Fanuc TP program (LS listing): MAKROSTP.LS

/PROG  MAKROSTP
/ATTR
OWNER		= MNEDITOR;
COMMENT		= "MAKRO_SCHRITT";
PROG_SIZE	= 100704;
CREATE		= DATE 11-01-11  TIME 07:00:00;
MODIFIED	= DATE 20-09-12  TIME 10:46:22;
FILE_NAME	= ;
VERSION		= 0;
LINE_COUNT	= 4405;
MEMORY_SIZE	= 103104;
PROTECT		= READ_WRITE;
TCD:  STACK_SIZE	= 0,
      TASK_PRIORITY	= 100,
      TIME_SLICE	= 0,
      BUSY_LAMP_OFF	= 1,
      ABORT_REQUEST	= 7,
      PAUSE_REQUEST	= 3;
DEFAULT_GROUP	= *,*,*,*,*;
CONTROL_CODE	= 00000000 00000010;
/MN
   1:  !Schrittkette Konzernstandard ;
   2:  !KS24 ;
   3:  !Version: 02 ;
   4:  !Stand: 003 MOD KN ;
   5:  !letzte Aenderung 30.07.2015 DB ;
   6:  !Mod von KN --> S2 mit Wartezeit ;
   7:   ;
   8:  !Zaehler [41] = aktueller Schritt ;
   9:  !Zaehler [42] = letzter Schritt ;
  10:  R[41]=0    ;
  11:  R[42]=0    ;
  12:   ;
  13:   ;
  14:  !*********************** ;
  15:  !*********************** ;
  16:  !* Start Makro_Schritt * ;
  17:  !*********************** ;
  18:  !*********************** ;
  19:   ;
  20:   ;
  21:  !***************************** ;
  22:  !*         Schritt 1         * ;
  23:  !* E/A's / Flags Ruecksetzen * ;
  24:  !***************************** ;
  25:   ;
  26:  !Loop fuer Schrittkette LBL[1] ;
  27:  LBL[1] ;
  28:  R[41]=1    ;
  29:  !Statusbildschirm einblenden ;
  30:  DO[18181]=(OFF) ;
  31:  !SK1 KF1 KS1 ;
  32:  DO[786]=(OFF) ;
  33:  DO[834]=(OFF) ;
  34:  DO[842]=(OFF) ;
  35:  DO[847]=(OFF) ;
  36:  !SK2 KF2 KS2 ;
  37:  DO[946]=(OFF) ;
  38:  DO[994]=(OFF) ;
  39:  DO[995]=(OFF) ;
  40:  DO[1002]=(OFF) ;
  41:  !SK3 KF3 KS3 ;
  42:  DO[1106]=(OFF) ;
  43:  DO[1154]=(OFF) ;
  44:  DO[1155]=(OFF) ;
  45:  DO[1162]=(OFF) ;
  46:  !KS1 KS2 KS3 ;
  47:  DO[3969]=(OFF) ;
  48:  DO[3970]=(OFF) ;
  49:  DO[3971]=(OFF) ;
  50:  !Auswahl EZ1/SP1 an KF2 ;
  51:  F[72]=(OFF) ;
  52:  !Auswahl EZ1/SP1 an KF3 ;
  53:  F[73]=(OFF) ;
  54:  !Auswert. KF Umdrehungen EZ1/SP1 ;
  55:  F[94]=(OFF) ;
  56:  F[95]=(OFF) ;
  57:  F[96]=(OFF) ;
  58:  F[97]=(OFF) ;
  59:  F[98]=(OFF) ;
  60:  F[99]=(OFF) ;
  61:  F[100]=(OFF) ;
  62:  F[101]=(OFF) ;
  63:  F[102]=(OFF) ;
  64:  F[103]=(OFF) ;
  65:  F[104]=(OFF) ;
  66:  F[105]=(OFF) ;
  67:  F[106]=(OFF) ;
  68:  F[107]=(OFF) ;
  69:  F[108]=(OFF) ;
  70:  F[109]=(OFF) ;
  71:  F[110]=(OFF) ;
  72:  F[111]=(OFF) ;
  73:  F[112]=(OFF) ;
  74:  F[113]=(OFF) ;
  75:  F[114]=(OFF) ;
  76:  F[115]=(OFF) ;
  77:  F[116]=(OFF) ;
  78:  F[117]=(OFF) ;
  79:  !Auswert. KF Umdrehungen EZ2/SP2 ;
  80:  F[150]=(OFF) ;
  81:  F[151]=(OFF) ;
  82:  F[152]=(OFF) ;
  83:  F[153]=(OFF) ;
  84:  F[154]=(OFF) ;
  85:  F[155]=(OFF) ;
  86:  !Auswert. KF Umdrehungen EZ3/SP3 ;
  87:  F[186]=(OFF) ;
  88:  F[187]=(OFF) ;
  89:  F[188]=(OFF) ;
  90:  F[189]=(OFF) ;
  91:  F[190]=(OFF) ;
  92:  F[191]=(OFF) ;
  93:  !Hilfsflags beim Fraesen ;
  94:  F[287]=(OFF) ;
  95:  F[290]=(OFF) ;
  96:  F[291]=(OFF) ;
  97:  F[301]=(OFF) ;
  98:  !Hilfsflags SZ2 an SK1 ;
  99:  F[307]=(OFF) ;
 100:  F[308]=(OFF) ;
 101:  !Hilfsflags KF Initiator ;
 102:  F[312]=(OFF) ;
 103:  F[313]=(OFF) ;
 104:  !RSK Fehlerausgaben ;
 105:  F[322]=(OFF) ;
 106:  F[323]=(OFF) ;
 107:  F[324]=(OFF) ;
 108:  F[325]=(OFF) ;
 109:  F[326]=(OFF) ;
 110:  F[327]=(OFF) ;
 111:  F[328]=(OFF) ;
 112:  F[329]=(OFF) ;
 113:  !Flag KL1 Spueleimer ;
 114:  F[352]=(OFF) ;
 115:  F[353]=(OFF) ;
 116:  !Flag KL2 Spueleimer ;
 117:  F[373]=(OFF) ;
 118:  F[374]=(OFF) ;
 119:  !Flag KL3 Spueleimer ;
 120:  F[394]=(OFF) ;
 121:  F[395]=(OFF) ;
 122:  !Flag MS Reinigung gestartet ;
 123:  F[604]=(OFF) ;
 124:  F[605]=(OFF) ;
 125:  F[608]=(OFF) ;
 126:  !Flag für Grundstellung RSK ;
 127:  F[321]=(OFF) ;
 128:  !Ruecksetzen Fraeszaehler ;
 129:  R[1]=0    ;
 130:  R[42]=1    ;
 131:  JMP LBL[2] ;
 132:   ;
 133:   ;
 134:  !************************ ;
 135:  !************************ ;
 136:  !* RSK in Grundstellung * ;
 137:  !************************ ;
 138:  !************************ ;
 139:   ;
 140:   ;
 141:  !*********************** ;
 142:  !*      Schritt 2      * ;
 143:  !* Funktionsauswertung * ;
 144:  !*********************** ;
 145:   ;
 146:  LBL[2] ;
 147:  R[41]=2    ;
 148:  F[321]=(ON) ;
 149:   ;
 150:  !Fraesen ROB EZ1/SP1 SZ1-SZ4 ;
 151:  !an KF1 ;
 152:  IF ((F[90] AND !F[91]) AND !F[72] AND !F[73] AND (F[64] OR F[65] OR F[66] OR F[67])),R[41]=3 ;
 153:   ;
 154:  !Fraesen ROB EZ1/SP1 SZ1-SZ4 ;
 155:  !an KF2 ;
 156:  IF ((F[90] AND !F[91]) AND F[72] AND !F[73] AND (F[64] OR F[65] OR F[66] OR F[67])),R[41]=58 ;
 157:   ;
 158:  !Fraesen ROB EZ1/SP1 SZ1-SZ4 ;
 159:  !an KF3 ;
 160:  IF ((F[90] AND !F[91]) AND !F[72] AND F[73] AND (F[64] OR F[65] OR F[66] OR F[67])),R[41]=64 ;
 161:   ;
 162:  !Fraesen STAT EZ1/SP1 ;
 163:  IF (F[92] AND !F[93]),R[41]=9 ;
 164:   ;
 165:  !Fraesen STAT EZ2/SP2 ;
 166:  IF (F[148] AND !F[149]),R[41]=18 ;
 167:   ;
 168:  !Fraesen STAT EZ3/SP3 ;
 169:  IF (F[184] AND !F[185]),R[41]=27 ;
 170:   ;
 171:  !MS1 Reinigung an KS3 ;
 172:  IF (F[603] AND !F[605] AND F[528] AND !F[529]),R[41]=36 ;
 173:   ;
 174:  !MS2 Reinigung an KS2 ;
 175:  IF (F[607] AND !F[609] AND F[528] AND !F[529]),R[41]=40 ;
 176:   ;
 177:  !KL1 Spueleimer (an Pneum. Schwen ;
 178:  !in Arbeitsstellung schwenken ;
 179:  IF (!F[352] AND F[353] AND !F[355] AND ((F[523] AND !F[524]) OR (!F[523] AND F[524]))),R[41]=44 ;
 180:   ;
 181:  !KL1 Spueleimer (an Pneum. Schwen ;
 182:  !in Ruhestellung schwenken ;
 183:  IF (F[352] AND !F[353] AND !F[355] AND ((F[523] AND !F[524]) OR (!F[523] AND F[524]))),R[41]=45 ;
 184:   ;
 185:  !KL2 Spueleimer (an Pneum. Schwen ;
 186:  !in Arbeitsstellung schwenken ;
 187:  IF (!F[373] AND F[374] AND !F[376] AND ((F[523] AND !F[524]) OR (!F[523] AND F[524]))),R[41]=46 ;
 188:   ;
 189:  !KL2 Spueleimer (an Pneum. Schwen ;
 190:  !in Ruhestellung schwenken ;
 191:  IF (F[373] AND !F[374] AND !F[376] AND ((F[523] AND !F[524]) OR (!F[523] AND F[524]))),R[41]=47 ;
 192:   ;
 193:  !KL3 Spueleimer (an Pneum. Schwen ;
 194:  !in Arbeitsstellung schwenken ;
 195:  IF (!F[394] AND F[395] AND !F[397] AND ((F[523] AND !F[524]) OR (!F[523] AND F[524]))),R[41]=48 ;
 196:   ;
 197:  !KL3 Spueleimer (an Pneum. Schwen ;
 198:  !in Ruhestellung schwenken ;
 199:  IF (F[394] AND !F[395] AND !F[397] AND ((F[523] AND !F[524]) OR (!F[523] AND F[524]))),R[41]=49 ;
 200:   ;
 201:  !MS1 Reinigung (an Pneum. Schwenk ;
 202:  IF (F[603] AND !F[605] AND !F[528] AND F[529]),R[41]=50 ;
 203:   ;
 204:  !Fraesen ROB STP SZ1 ;
 205:  IF (F[64] AND !F[65] AND !F[66] AND !F[67] AND F[90] AND !F[91] AND F[565]),R[41]=70 ;
 206:   ;
 207:  !Wartezeit fuer Synconisation ;
 208:  WAIT    .20(sec) ;
 209:   ;
 210:  R[42]=2    ;
 211:  JMP LBL[R[41]] ;
 212:   ;
 213:   ;
 214:  !*************************** ;
 215:  !*************************** ;
 216:  !* Fraesen Rob EZ1 SZ1-SZ4 * ;
 217:  !*          an KF1         * ;
 218:  !*************************** ;
 219:  !*************************** ;
 220:   ;
 221:   ;
 222:  !**************************** ;
 223:  !*        Schritt 3         * ;
 224:  !* Rob EZ1 SZ1-SZ4 Auswert. * ;
 225:  !**************************** ;
 226:   ;
 227:  LBL[3] ;
 228:  R[41]=3    ;
 229:  !RSK gestartet ;
 230:  F[321]=(OFF) ;
 231:  GO[1]=(31) ;
 232:  IF (F[64]),GO[3]=(31) ;
 233:  IF (F[65]),GO[3]=(32) ;
 234:  IF (F[66]),GO[3]=(33) ;
 235:  IF (F[67]),GO[3]=(34) ;
 236:  WAIT    .10(sec) ;
 237:  DO[116]=(ON) ;
 238:  DO[130]=(ON) ;
 239:  DO[718]=(OFF) ;
 240:  DO[717]=(!DI[717]) ;
 241:  DO[18181]=(ON) ;
 242:  WAIT (DI[717])    ;
 243:  DO[18181]=(OFF) ;
 244:  DO[717]=(OFF) ;
 245:  !Anwahl Startfraesen ;
 246:  IF (F[90] AND F[78] AND !F[79]),R[41]=4 ;
 247:  !Anwahl Normalfraesen ;
 248:  IF (F[90] AND !F[78] AND F[79]),R[41]=6 ;
 249:  R[42]=3    ;
 250:  JMP LBL[R[41]] ;
 251:   ;
 252:  !***************************** ;
 253:  !*         Schritt 4         * ;
 254:  !* Rob EZ1 SZ1-SZ4 SF Teil 1 * ;
 255:  !***************************** ;
 256:   ;
 257:  LBL[4] ;
 258:  R[41]=4    ;
 259:  !RSK gestartet ;
 260:  F[321]=(OFF) ;
 261:  F[329]=(OFF) ;
 262:  F[325]=(OFF) ;
 263:  DO[718]=(OFF) ;
 264:  DO[717]=(!DI[717]) ;
 265:  DO[18181]=(ON) ;
 266:  WAIT (DI[717])    ;
 267:  DO[18181]=(OFF) ;
 268:  DO[834]=(ON) ;
 269:  DO[858]=(ON) ;
 270:  DO[835]=(F[330]) ;
 271:  DO[859]=(F[330]) ;
 272:  DO[717]=(OFF) ;
 273:  !Warte Fraeser laeuft ;
 274:  TIMER[7]=((-3)) ;
 275:  WAIT ((!DI[834] AND !F[289]) OR (!DI[858] AND F[289]) OR (TIMER[7]>=0))    ;
 276:  WAIT ((DI[834] AND !F[289]) OR (DI[858] AND F[289]) OR (TIMER[7]>=0))    ;
 277:  F[322]=((TIMER[7]>=0)) ;
 278:  DO[18181]=(ON) ;
 279:  WAIT ((!DI[834] AND !F[289]) OR (!DI[858] AND F[289]))    ;
 280:  WAIT ((DI[834] AND !F[289]) OR (DI[858] AND F[289]))    ;
 281:  DO[18181]=(OFF) ;
 282:  F[322]=(OFF) ;
 283:  !EZ1/SP1 schliessen ;
 284:  DO[718]=(ON) ;
 285:  TIMER[9]=((-4)) ;
 286:  !EZ1/SP1 Kraft erreicht ;
 287:  WAIT ((DI[718] AND !DI[772] AND !DI[780] AND !DI[774] AND !DI[775]) OR (TIMER[9]>=0))    ;
 288:  DO[18181]=(ON) ;
 289:  DO[718]=((TIMER[9]<0)) ;
 290:  DO[834]=((TIMER[9]<0)) ;
 291:  DO[858]=((TIMER[9]<0)) ;
 292:  WAIT ((DI[718] AND !DI[772] AND !DI[780] AND !DI[774] AND !DI[775]) OR DI[26] OR DI[27])    ;
 293:  F[325]=(DI[26] OR DI[27]) ;
 294:  DO[18181]=(OFF) ;
 295:  !EZ1/SP1 Fehler Kraftaufbau ;
 296:  IF (F[325]),JMP LBL[406] ;
 297:  TIMER[9]=((-5)) ;
 298:  LBL[400] ;
 299:  WAIT ((!DI[834] AND !F[289]) OR (!DI[858] AND F[289]) OR F[325] OR (TIMER[9]>=0))    ;
 300:  WAIT ((DI[834] AND !F[289]) OR (DI[858] AND F[289]) OR F[325] OR (TIMER[9]>=0))    ;
 301:  R[1]=(R[1]+1) ;
 302:  F[329]=((TIMER[9]>=0)) ;
 303:  !Fraeszeit ueberschritten ;
 304:  IF (F[329]),JMP LBL[406] ;
 305:  IF (F[64]),JMP LBL[402] ;
 306:  IF (F[65]),JMP LBL[403] ;
 307:  IF (F[66]),JMP LBL[404] ;
 308:  IF (F[67]),JMP LBL[405] ;
 309:  !Umdrehungen Vergl.SZ1 ;
 310:  LBL[402] ;
 311:  !Umdrehungen Vergleichen ;
 312:  IF (R[1]<R[2]),JMP LBL[400] ;
 313:  JMP LBL[401] ;
 314:  !Umdrehungen Vergl.SZ2 ;
 315:  LBL[403] ;
 316:  !Umdrehungen Vergleichen ;
 317:  IF (R[1]<R[8]),JMP LBL[400] ;
 318:  JMP LBL[401] ;
 319:  !Umdrehungen Vergl.SZ3 ;
 320:  LBL[404] ;
 321:  !Umdrehungen Vergleichen ;
 322:  IF (R[1]<R[11]),JMP LBL[400] ;
 323:  JMP LBL[401] ;
 324:  !Umdrehungen Vergl.SZ4 ;
 325:  LBL[405] ;
 326:  !Umdrehungen Vergleichen ;
 327:  IF (R[1]<R[14]),JMP LBL[400] ;
 328:  JMP LBL[401] ;
 329:  LBL[401] ;
 330:  IF (F[64]),F[94]=(ON) ;
 331:  IF (F[65]),F[100]=(ON) ;
 332:  IF (F[66]),F[106]=(ON) ;
 333:  IF (F[67]),F[112]=(ON) ;
 334:  LBL[406] ;
 335:  DO[834]=((TIMER[9]<0)) ;
 336:  DO[858]=((TIMER[9]<0)) ;
 337:  !Fraeser ausblasen EIN ;
 338:  DO[835]=(F[330] OR (TIMER[9]<0)) ;
 339:  DO[859]=(F[330] OR (TIMER[9]<0)) ;
 340:  DO[718]=(OFF) ;
 341:  !EZ1/SP1 oeffnen ;
 342:  DO[717]=(!DI[717]) ;
 343:  DO[18181]=(F[329]) ;
 344:  WAIT (!F[329] OR DI[26] OR DI[27])    ;
 345:  DO[18181]=(OFF) ;
 346:  DO[18181]=(ON) ;
 347:  WAIT (DI[717])    ;
 348:  DO[18181]=(OFF) ;
 349:  DO[717]=(OFF) ;
 350:  !Umdrehungen ruecksetzen ;
 351:  R[1]=0    ;
 352:  R[42]=4    ;
 353:  IF (F[329] OR F[325]),JMP LBL[4] ;
 354:  JMP LBL[5] ;
 355:   ;
 356:  !***************************** ;
 357:  !*         Schritt 5         * ;
 358:  !* Rob EZ1 SZ1-SZ4 SF Teil 2 * ;
 359:  !***************************** ;
 360:   ;
 361:  LBL[5] ;
 362:  R[41]=5    ;
 363:  !RSK gestartet ;
 364:  F[321]=(OFF) ;
 365:  F[329]=(OFF) ;
 366:  F[325]=(OFF) ;
 367:  DO[718]=(OFF) ;
 368:  DO[717]=(!DI[717]) ;
 369:  DO[18181]=(ON) ;
 370:  WAIT (DI[717])    ;
 371:  DO[18181]=(OFF) ;
 372:  DO[834]=(ON) ;
 373:  DO[858]=(ON) ;
 374:  DO[717]=(OFF) ;
 375:  !EZ1/SP1 schliessen ;
 376:  DO[718]=(ON) ;
 377:  !Fraeser ausblasen AUS/AN ;
 378:  DO[835]=(F[330]) ;
 379:  DO[859]=(F[330]) ;
 380:  TIMER[9]=((-4)) ;
 381:  !EZ1/SP1 Kraft erreicht ;
 382:  WAIT ((DI[718] AND !DI[772] AND !DI[780] AND !DI[774] AND !DI[775]) OR (TIMER[9]>=0))    ;
 383:  DO[18181]=(ON) ;
 384:  DO[718]=((TIMER[9]<0)) ;
 385:  DO[834]=((TIMER[9]<0)) ;
 386:  DO[858]=((TIMER[9]<0)) ;
 387:  WAIT ((DI[718] AND !DI[772] AND !DI[780] AND !DI[774] AND !DI[775]) OR DI[26] OR DI[27])    ;
 388:  F[325]=(DI[26] OR DI[27]) ;
 389:  DO[18181]=(OFF) ;
 390:  !EZ1/SP1 Fehler Kraftaufbau ;
 391:  IF (F[325]),JMP LBL[5] ;
 392:  TIMER[9]=((-5)) ;
 393:  LBL[500] ;
 394:  WAIT ((!DI[834] AND !F[289]) OR (!DI[858] AND F[289]) OR F[325] OR (TIMER[9]>=0))    ;
 395:  WAIT ((DI[834] AND !F[289]) OR (DI[858] AND F[289]) OR F[325] OR (TIMER[9]>=0))    ;
 396:  R[1]=(R[1]+1) ;
 397:  F[329]=((TIMER[9]>=0)) ;
 398:  !Fraeszeit ueberschritten ;
 399:  IF (F[329]),JMP LBL[506] ;
 400:  IF (F[64]),JMP LBL[502] ;
 401:  IF (F[65]),JMP LBL[503] ;
 402:  IF (F[66]),JMP LBL[504] ;
 403:  IF (F[67]),JMP LBL[505] ;
 404:  !Umdrehungen Vergl.SZ1 ;
 405:  LBL[502] ;
 406:  !Umdrehungen Vergleichen ;
 407:  IF (R[1]<R[3]),JMP LBL[500] ;
 408:  JMP LBL[501] ;
 409:  !Umdrehungen Vergl.SZ2 ;
 410:  LBL[503] ;
 411:  !Umdrehungen Vergleichen ;
 412:  IF (R[1]<R[9]),JMP LBL[500] ;
 413:  JMP LBL[501] ;
 414:  !Umdrehungen Vergl.SZ3 ;
 415:  LBL[504] ;
 416:  !Umdrehungen Vergleichen ;
 417:  IF (R[1]<R[12]),JMP LBL[500] ;
 418:  JMP LBL[501] ;
 419:  !Umdrehungen Vergl.SZ4 ;
 420:  LBL[505] ;
 421:  !Umdrehungen Vergleichen ;
 422:  IF (R[1]<R[15]),JMP LBL[500] ;
 423:  JMP LBL[501] ;
 424:  LBL[501] ;
 425:  IF (F[64]),F[96]=(ON) ;
 426:  IF (F[65]),F[102]=(ON) ;
 427:  IF (F[66]),F[108]=(ON) ;
 428:  IF (F[67]),F[114]=(ON) ;
 429:  LBL[506] ;
 430:  DO[834]=((TIMER[9]<0)) ;
 431:  DO[858]=((TIMER[9]<0)) ;
 432:  !Fraeser ausblasen EIN ;
 433:  DO[835]=PULSE,4.0sec ;
 434:  DO[859]=PULSE,4.0sec ;
 435:  DO[718]=(OFF) ;
 436:  !EZ1/SP1 oeffnen ;
 437:  DO[717]=(!DI[717]) ;
 438:  DO[18181]=(F[329]) ;
 439:  WAIT (!F[329] OR DI[26] OR DI[27])    ;
 440:  DO[18181]=(OFF) ;
 441:  DO[18181]=(ON) ;
 442:  WAIT (DI[717])    ;
 443:  DO[18181]=(OFF) ;
 444:  DO[717]=(OFF) ;
 445:  !Umdrehungen ruecksetzen ;
 446:  R[1]=0    ;
 447:  R[42]=5    ;
 448:  IF (F[329] OR F[325]),JMP LBL[5] ;
 449:  JMP LBL[7] ;
 450:   ;
 451:  !********************** ;
 452:  !*     Schritt 6      * ;
 453:  !* Rob EZ1 SZ1-SZ4 NF * ;
 454:  !********************** ;
 455:   ;
 456:  LBL[6] ;
 457:  R[41]=6    ;
 458:  !RSK gestartet ;
 459:  F[321]=(OFF) ;
 460:  F[329]=(OFF) ;
 461:  F[325]=(OFF) ;
 462:  !Zähler wegspeichern für 2ten Hub ;
 463:  R[45]=R[4]    ;
 464:  IF (F[98] AND F[732]),R[4]=R[43] ;
 465:  !Überprüfungung Zangenstellung ;
 466:  DO[718]=(OFF) ;
 467:  DO[717]=(!DI[717]) ;
 468:  DO[18181]=(ON) ;
 469:  WAIT (DI[717])    ;
 470:  DO[18181]=(OFF) ;
 471:  DO[834]=(ON) ;
 472:  DO[835]=(F[330]) ;
 473:  DO[858]=(ON) ;
 474:  DO[859]=(F[330]) ;
 475:  DO[717]=(OFF) ;
 476:  !Warte Fraeser laeuft ;
 477:  TIMER[7]=((-3)) ;
 478:  WAIT ((!DI[834] AND !F[289]) OR (!DI[858] AND F[289]) OR (TIMER[7]>=0))    ;
 479:  WAIT ((DI[834] AND !F[289]) OR (DI[858] AND F[289]) OR (TIMER[7]>=0))    ;
 480:  F[322]=((TIMER[7]>=0)) ;
 481:  DO[18181]=(ON) ;
 482:  WAIT ((!DI[834] AND !F[289]) OR (!DI[858] AND F[289]))    ;
 483:  WAIT ((DI[834] AND !F[289]) OR (DI[858] AND F[289]))    ;
 484:  DO[18181]=(OFF) ;
 485:  F[322]=(OFF) ;
 486:  !EZ1/SP1 schliessen ;
 487:  DO[718]=(ON) ;
 488:  TIMER[9]=((-4)) ;
 489:  !EZ1/SP1 Kraft erreicht ;
 490:  WAIT ((DI[718] AND !DI[772] AND !DI[780] AND !DI[774] AND !DI[775]) OR (TIMER[9]>=0))    ;
 491:  DO[18181]=(ON) ;
 492:  DO[718]=((TIMER[9]<0)) ;
 493:  DO[834]=((TIMER[9]<0)) ;
 494:  DO[858]=((TIMER[9]<0)) ;
 495:  WAIT ((DI[718] AND !DI[772] AND !DI[780] AND !DI[774] AND !DI[775]) OR DI[26] OR DI[27])    ;
 496:  F[325]=(DI[26] OR DI[27]) ;
 497:  DO[18181]=(OFF) ;
 498:  !EZ1/SP1 Fehler Kraftaufbau ;
 499:  IF (F[325]),JMP LBL[6] ;
 500:  TIMER[9]=((-5)) ;
 501:  LBL[600] ;
 502:  WAIT ((!DI[834] AND !F[289]) OR (!DI[858] AND F[289]) OR F[325] OR (TIMER[9]>=0))    ;
 503:  WAIT ((DI[834] AND !F[289]) OR (DI[858] AND F[289]) OR F[325] OR (TIMER[9]>=0))    ;
 504:  R[1]=(R[1]+1) ;
 505:  F[329]=((TIMER[9]>=0)) ;
 506:  !Fraeszeit ueberschritten ;
 507:  IF (F[329]),JMP LBL[606] ;
 508:  IF (F[64]),JMP LBL[602] ;
 509:  IF (F[65]),JMP LBL[603] ;
 510:  IF (F[66]),JMP LBL[604] ;
 511:  IF (F[67]),JMP LBL[605] ;
 512:  !Umdrehungen Vergl.SZ1 ;
 513:  LBL[602] ;
 514:  !Umdrehungen Vergleichen ;
 515:  IF (R[1]<R[4]),JMP LBL[600] ;
 516:  JMP LBL[601] ;
 517:  !Umdrehungen Vergl.SZ2 ;
 518:  LBL[603] ;
 519:  !Umdrehungen Vergleichen ;
 520:  IF (R[1]<R[10]),JMP LBL[600] ;
 521:  !Umdrehungen Vergl.SZ3 ;
 522:  LBL[604] ;
 523:  !Umdrehungen Vergleichen ;
 524:  IF (R[1]<R[13]),JMP LBL[600] ;
 525:  JMP LBL[601] ;
 526:  !Umdrehungen Vergl.SZ4 ;
 527:  LBL[605] ;
 528:  !Umdrehungen Vergleichen ;
 529:  IF (R[1]<R[16]),JMP LBL[600] ;
 530:  LBL[601] ;
 531:  !EZ1/SP1 2 Huebe bei NF ;
 532:  IF (!F[130]),JMP LBL[606] ;
 533:  IF (F[98]),F[96]=(ON) ;
 534:  IF (F[104]),F[96]=(ON) ;
 535:  IF (F[110]),F[96]=(ON) ;
 536:  IF (F[116]),F[96]=(ON) ;
 537:  IF (F[64]),F[98]=(ON) ;
 538:  IF (F[65]),F[104]=(ON) ;
 539:  IF (F[66]),F[110]=(ON) ;
 540:  IF (F[67]),F[116]=(ON) ;
 541:  LBL[606] ;
 542:  DO[834]=((TIMER[9]<0)) ;
 543:  DO[858]=((TIMER[9]<0)) ;
 544:  !Fraeser ausblasen EIN ;
 545:  DO[835]=PULSE,4.0sec ;
 546:  DO[859]=PULSE,4.0sec ;
 547:  DO[718]=(OFF) ;
 548:  !EZ1/SP1 oeffnen ;
 549:  DO[717]=(!DI[717]) ;
 550:  DO[18181]=(F[329]) ;
 551:  WAIT (!F[329] OR DI[26] OR DI[27])    ;
 552:  DO[18181]=(OFF) ;
 553:  DO[18181]=(ON) ;
 554:  WAIT (DI[717])    ;
 555:  DO[18181]=(OFF) ;
 556:  DO[717]=(OFF) ;
 557:  !Umdrehungen ruecksetzen ;
 558:  R[1]=0    ;
 559:  R[42]=6    ;
 560:  !Zähler umschreiben für 2ten Hub ;
 561:  IF (F[98] AND F[732] AND F[64]),GO[3]=36 ;
 562:  IF (F[104] AND F[732] AND F[65]),GO[3]=37 ;
 563:  IF (F[110] AND F[732] AND F[66]),GO[3]=38 ;
 564:  IF (F[116] AND F[732] AND F[67]),GO[3]=39 ;
 565:  IF (F[96] AND F[732]),R[4]=R[45] ;
 566:  !Aufruf 2ter Hub ;
 567:  IF (F[329] OR (!F[96] AND F[130])),JMP LBL[6] ;
 568:  IF (F[64]),F[98]=(ON) ;
 569:  IF (F[65]),F[104]=(ON) ;
 570:  IF (F[66]),F[110]=(ON) ;
 571:  IF (F[67]),F[116]=(ON) ;
 572:  JMP LBL[7] ;
 573:   ;
 574:  !******************************* ;
 575:  !*         Schritt 7           * ;
 576:  !* Rob EZ1 SZ1-SZ4 i.O./n.i.O. * ;
 577:  !******************************* ;
 578:   ;
 579:  LBL[7] ;
 580:  R[41]=7    ;
 581:  !Fraesueberwachung starten ;
 582:  IF (F[64]),JMP LBL[701] ;
 583:  IF (F[65]),JMP LBL[702] ;
 584:  IF (F[66]),JMP LBL[703] ;
 585:  IF (F[67]),JMP LBL[704] ;
 586:  LBL[701] ;
 587:  TIMER[7]=((-3)) ;
 588:  WAIT (F[64] AND ((F[79] AND F[98]) OR (F[78] AND F[94] AND F[96])) OR (TIMER[7]>=0))    ;
 589:  F[329]=((TIMER[7]>=0)) ;
 590:  DO[18181]=(ON) ;
 591:  WAIT (F[64] AND ((F[79] AND F[98]) OR (F[78] AND F[94] AND F[96])))    ;
 592:  DO[18181]=(OFF) ;
 593:  JMP LBL[700] ;
 594:  LBL[702] ;
 595:  TIMER[7]=((-3)) ;
 596:  WAIT (F[65] AND ((F[79] AND F[104]) OR (F[78] AND F[100] AND F[102])) OR (TIMER[7]>=0))    ;
 597:  F[329]=((TIMER[7]>=0)) ;
 598:  DO[18181]=(ON) ;
 599:  WAIT (F[65] AND ((F[79] AND F[104]) OR (F[78] AND F[100] AND F[102])))    ;
 600:  DO[18181]=(OFF) ;
 601:  JMP LBL[700] ;
 602:  LBL[703] ;
 603:  TIMER[7]=((-3)) ;
 604:  WAIT (F[66] AND ((F[79] AND F[110]) OR (F[78] AND F[106] AND F[108])) OR (TIMER[7]>=0))    ;
 605:  F[329]=((TIMER[7]>=0)) ;
 606:  DO[18181]=(ON) ;
 607:  WAIT (F[66] AND ((F[79] AND F[110]) OR (F[78] AND F[106] AND F[108])))    ;
 608:  DO[18181]=(OFF) ;
 609:  JMP LBL[700] ;
 610:  LBL[704] ;
 611:  TIMER[7]=((-3)) ;
 612:  WAIT (F[67] AND ((F[79] AND F[116]) OR (F[78] AND F[112] AND F[114])) OR (TIMER[7]>=0))    ;
 613:  F[329]=((TIMER[7]>=0)) ;
 614:  DO[18181]=(ON) ;
 615:  WAIT (F[67] AND ((F[79] AND F[116]) OR (F[78] AND F[112] AND F[114])))    ;
 616:  DO[18181]=(OFF) ;
 617:  JMP LBL[700] ;
 618:  LBL[700] ;
 619:  R[41]=8    ;
 620:  !KF1 U-Merker ruecksetzen ;
 621:  F[94]=(OFF) ;
 622:  F[96]=(OFF) ;
 623:  F[98]=(OFF) ;
 624:  F[100]=(OFF) ;
 625:  F[102]=(OFF) ;
 626:  F[104]=(OFF) ;
 627:  F[106]=(OFF) ;
 628:  F[108]=(OFF) ;
 629:  F[110]=(OFF) ;
 630:  F[112]=(OFF) ;
 631:  F[114]=(OFF) ;
 632:  F[116]=(OFF) ;
 633:  R[42]=7    ;
 634:  JMP LBL[R[41]] ;
 635:   ;
 636:  !***************************** ;
 637:  !*        Schritt 8          * ;
 638:  !* Rob EZ1 SZ1-SZ4 Quitt SK1 * ;
 639:  !***************************** ;
 640:   ;
 641:  LBL[8] ;
 642:  R[41]=8    ;
 643:  !RSK gestartet ;
 644:  F[321]=(OFF) ;
 645:  IF (F[64]),GO[3]=1 ;
 646:  IF (F[65]),GO[3]=2 ;
 647:  IF (F[66]),GO[3]=3 ;
 648:  IF (F[67]),GO[3]=4 ;
 649:  WAIT    .10(sec) ;
 650:  DO[786]=(ON) ;
 651:  DO[116]=(OFF) ;
 652:  DO[130]=(OFF) ;
 653:  DO[18181]=(ON) ;
 654:  WAIT (!DI[786] AND DI[787] AND !DI[788])    ;
 655:  !FK Fraesen ;
 656:  F[91]=(!F[329]) ;
 657:  DO[18181]=(OFF) ;
 658:  DO[786]=(OFF) ;
 659:  R[42]=8    ;
 660:  JMP LBL[1] ;
 661:   ;
 662:   ;
 663:  !************************ ;
 664:  !************************ ;
 665:  !* Fraesen STAT EZ1/SP1 * ;
 666:  !************************ ;
 667:  !************************ ;
 668:   ;
 669:   ;
 670:  !****************************** ;
 671:  !*         Schritt 9          * ;
 672:  !*        STAT EZ1/SP1        * ;
 673:  !* KS1 in Arbeitsst.schwenken * ;
 674:  !****************************** ;
 675:   ;
 676:  LBL[9] ;
 677:  R[41]=9    ;
 678:  !RSK gestartet ;
 679:  F[321]=(OFF) ;
 680:  GO[1]=(31) ;
 681:  GO[3]=(31) ;
 682:  WAIT    .10(sec) ;
 683:  DO[758]=(F[78]) ;
 684:  DO[759]=(F[79]) ;
 685:  DO[116]=(ON) ;
 686:  DO[130]=(ON) ;
 687:  DO[718]=(OFF) ;
 688:  DO[717]=(!DI[717]) ;
 689:  DO[18181]=(ON) ;
 690:  WAIT (DI[717])    ;
 691:  DO[18181]=(OFF) ;
 692:  DO[717]=(OFF) ;
 693:  !Ueberwachungszeit Grundstellung ;
 694:  TIMER[8]=((-4)) ;
 695:  WAIT ((DI[842] AND !DI[843] AND !DI[844] AND DI[845]) OR (TIMER[8]>=0))    ;
 696:  F[323]=((TIMER[8]>=0)) ;
 697:  DO[18181]=((TIMER[8]>=0)) ;
 698:  WAIT (DI[842] AND !DI[843] AND !DI[844] AND DI[845])    ;
 699:  DO[18181]=(OFF) ;
 700:  F[323]=(OFF) ;
 701:  TIMER[8]=((-4)) ;
 702:  DO[835]=(F[564]) ;
 703:  WAIT ((DI[835] AND F[564]) OR (!DI[835] AND !F[564]) OR (TIMER[8]>=0))    ;
 704:  F[323]=((TIMER[8]>=0)) ;
 705:  DO[18181]=((TIMER[8]>=0)) ;
 706:  WAIT ((DI[835] AND F[564]) OR (!DI[835] AND !F[564]))    ;
 707:  DO[18181]=(OFF) ;
 708:  F[323]=(OFF) ;
 709:  !Ueberwachungszeit KS1 Schwenken ;
 710:  TIMER[8]=((-6)) ;
 711:  !KS1 in Arbeitst. schwenken ;
 712:  DO[3972]=(ON) ;
 713:  WAIT (DI[841] OR (TIMER[8]>=0))    ;
 714:  DO[18181]=((TIMER[8]>=0)) ;
 715:  WAIT (DI[841])    ;
 716:  TIMER[8]=((-6)) ;
 717:  DO[18181]=(OFF) ;
 718:  WAIT ((!DI[842] AND DI[843] AND DI[844] AND !DI[845]) OR (TIMER[8]>=0))    ;
 719:  F[324]=((TIMER[8]>=0)) ;
 720:  DO[3972]=(OFF) ;
 721:  DO[18181]=((TIMER[8]>=0)) ;
 722:  WAIT ((!DI[842] AND DI[843] AND DI[844] AND !DI[845]) OR DI[26])    ;
 723:  DO[18181]=(OFF) ;
 724:  F[324]=(OFF) ;
 725:  !Sprung zurueck bei KS1 Fehler ;
 726:  IF (TIMER[8]>=0),JMP LBL[9] ;
 727:  DO[835]=(OFF) ;
 728:  TIMER[11]=((R[24])) ;
 729:  WAIT ((TIMER[11]>=0) OR !F[564])    ;
 730:  TIMER[11]=STOP ;
 731:  DO[18181]=(ON) ;
 732:  WAIT ((F[92] AND F[78]) OR (F[92] AND F[79]))    ;
 733:  DO[18181]=(OFF) ;
 734:  !Anwahl Startfraesen ;
 735:  IF (!DI[842] AND DI[843] AND F[92] AND F[78] AND !F[301]),R[41]=10 ;
 736:  !Anwahl Normalfraesen ;
 737:  IF (!DI[842] AND DI[843] AND F[92] AND (F[79] OR F[301])),R[41]=12 ;
 738:  R[42]=9    ;
 739:  JMP LBL[R[41]] ;
 740:   ;
 741:  !************************** ;
 742:  !*       Schritt 10       * ;
 743:  !* STAT EZ1/SP1 SF Teil 1 * ;
 744:  !************************** ;
 745:   ;
 746:  LBL[10] ;
 747:  R[41]=10    ;
 748:  !RSK gestartet ;
 749:  F[321]=(OFF) ;
 750:  F[329]=(OFF) ;
 751:  F[325]=(OFF) ;
 752:  DO[718]=(OFF) ;
 753:  DO[717]=(!DI[717]) ;
 754:  DO[18181]=(ON) ;
 755:  WAIT (DI[717])    ;
 756:  DO[717]=(OFF) ;
 757:  DO[18181]=(OFF) ;
 758:  DO[834]=(ON) ;
 759:  !Warte Fraeser laeuft ;
 760:  TIMER[7]=((-3)) ;
 761:  WAIT (!DI[834] OR (TIMER[7]>=0))    ;
 762:  WAIT (DI[834] OR (TIMER[7]>=0))    ;
 763:  F[322]=((TIMER[7]>=0)) ;
 764:  DO[18181]=(ON) ;
 765:  WAIT (!DI[834])    ;
 766:  WAIT (DI[834])    ;
 767:  DO[18181]=(OFF) ;
 768:  F[322]=(OFF) ;
 769:  !EZ1/SP1 schliessen ;
 770:  DO[718]=(ON) ;
 771:  !Fraeser ausblasen AUS/EIN ;
 772:  DO[847]=(F[330]) ;
 773:  TIMER[9]=((-4)) ;
 774:  !EZ1/SP1 Kraft erreicht ;
 775:  WAIT ((DI[718] AND !DI[772] AND !DI[780] AND !DI[774] AND !DI[775]) OR (TIMER[9]>=0))    ;
 776:  F[325]=((TIMER[9]>=0)) ;
 777:  DO[18181]=(ON) ;
 778:  DO[718]=((TIMER[9]<0)) ;
 779:  DO[834]=((TIMER[9]<0)) ;
 780:  WAIT ((DI[718] AND !DI[772] AND !DI[780] AND !DI[774] AND !DI[775]) OR DI[26] OR DI[27])    ;
 781:  DO[18181]=(OFF) ;
 782:  !EZ1/SP1 Fehler Kraftaufbau ;
 783:  IF (F[325]),JMP LBL[1001] ;
 784:  TIMER[9]=((-5)) ;
 785:  LBL[1000] ;
 786:  WAIT (!DI[834] OR F[325] OR (TIMER[9]>=0))    ;
 787:  WAIT (DI[834] OR F[325] OR (TIMER[9]>=0))    ;
 788:  R[1]=(R[1]+1) ;
 789:  F[329]=((TIMER[9]>=0)) ;
 790:  !Fraeszeit ueberschritten ;
 791:  IF (F[329]),JMP LBL[1001] ;
 792:  !Umdrehungen Vergleichen ;
 793:  IF (R[1]<R[2]),JMP LBL[1000] ;
 794:  F[94]=(ON) ;
 795:  LBL[1001] ;
 796:  DO[834]=((TIMER[9]<0)) ;
 797:  !Fraeser ausblasen EIN ;
 798:  DO[847]=(F[330] OR (TIMER[9]<0)) ;
 799:  DO[718]=(OFF) ;
 800:  !EZ1/SP1 oeffnen ;
 801:  DO[717]=(!DI[717]) ;
 802:  DO[18181]=(F[329]) ;
 803:  WAIT (!F[329] OR DI[26] OR DI[27])    ;
 804:  DO[18181]=(OFF) ;
 805:  DO[18181]=(ON) ;
 806:  WAIT (DI[717])    ;
 807:  DO[18181]=(OFF) ;
 808:  DO[717]=(OFF) ;
 809:  !Umdrehungen ruecksetzen ;
 810:  R[1]=0    ;
 811:  R[42]=10    ;
 812:  IF (F[329] OR F[325]),JMP LBL[10] ;
 813:  JMP LBL[11] ;
 814:   ;
 815:  !************************** ;
 816:  !*       Schritt 11       * ;
 817:  !* STAT EZ1/SP1 SF Teil 2 * ;
 818:  !************************** ;
 819:   ;
 820:  LBL[11] ;
 821:  R[41]=11    ;
 822:  !RSK gestartet ;
 823:  F[321]=(OFF) ;
 824:  F[329]=(OFF) ;
 825:  F[325]=(OFF) ;
 826:  DO[718]=(OFF) ;
 827:  DO[717]=(!DI[717]) ;
 828:  DO[18181]=(ON) ;
 829:  WAIT (DI[717])    ;
 830:  DO[18181]=(OFF) ;
 831:  DO[834]=(ON) ;
 832:  DO[717]=(OFF) ;
 833:  !EZ1/SP1 schliessen ;
 834:  DO[718]=(ON) ;
 835:  !Fraeser ausblasen AUS/EIN ;
 836:  DO[847]=(F[330]) ;
 837:  TIMER[9]=((-4)) ;
 838:  !EZ1/SP1 Kraft erreicht ;
 839:  WAIT ((DI[718] AND !DI[772] AND !DI[780] AND !DI[774] AND !DI[775]) OR (TIMER[9]>=0))    ;
 840:  F[325]=((TIMER[9]>=0)) ;
 841:  DO[18181]=(ON) ;
 842:  DO[718]=((TIMER[9]<0)) ;
 843:  DO[834]=((TIMER[9]<0)) ;
 844:  WAIT ((DI[718] AND !DI[772] AND !DI[780] AND !DI[774] AND !DI[775]) OR DI[26] OR DI[27])    ;
 845:  DO[18181]=(OFF) ;
 846:  !EZ1/SP1 Fehler Kraftaufbau ;
 847:  IF (F[325]),JMP LBL[1101] ;
 848:  TIMER[9]=((-5)) ;
 849:  LBL[1100] ;
 850:  WAIT (!DI[834] OR F[325] OR (TIMER[9]>=0))    ;
 851:  WAIT (DI[834] OR F[325] OR (TIMER[9]>=0))    ;
 852:  R[1]=(R[1]+1) ;
 853:  F[329]=((TIMER[9]>=0)) ;
 854:  !Fraeszeit ueberschritten ;
 855:  IF (F[329]),JMP LBL[1101] ;
 856:  !Umdrehungen Vergleichen ;
 857:  IF (R[1]<R[3]),JMP LBL[1100] ;
 858:  F[96]=(ON) ;
 859:  LBL[1101] ;
 860:  DO[834]=((TIMER[9]<0)) ;
 861:  !Fraeser ausblasen EIN ;
 862:  DO[847]=PULSE,4.0sec ;
 863:  DO[718]=(OFF) ;
 864:  !EZ1/SP1 oeffnen ;
 865:  DO[717]=(!DI[717]) ;
 866:  DO[18181]=(F[329]) ;
 867:  WAIT (!F[329] OR DI[26] OR DI[27])    ;
 868:  DO[18181]=(OFF) ;
 869:  DO[18181]=(ON) ;
 870:  WAIT (DI[717])    ;
 871:  DO[18181]=(OFF) ;
 872:  DO[717]=(OFF) ;
 873:  !Umdrehungen ruecksetzen ;
 874:  R[1]=0    ;
 875:  R[42]=11    ;
 876:  IF (F[329] OR F[325]),JMP LBL[11] ;
 877:  JMP LBL[13] ;
 878:   ;
 879:  !******************* ;
 880:  !*   Schritt 12    * ;
 881:  !* STAT EZ1/SP1 NF * ;
 882:  !******************* ;
 883:   ;
 884:  LBL[12] ;
 885:  R[41]=12    ;
 886:  !RSK gestartet ;
 887:  F[321]=(OFF) ;
 888:  F[329]=(OFF) ;
 889:  F[325]=(OFF) ;
 890:  !Zähler wegspeichern für 2ten Hub ;
 891:  R[45]=R[4]    ;
 892:  IF (F[98] AND F[732]),R[4]=R[43] ;
 893:  !Überprüfungung Zangenstellung ;
 894:  DO[718]=(OFF) ;
 895:  DO[717]=(!DI[717]) ;
 896:  DO[18181]=(ON) ;
 897:  WAIT (DI[717])    ;
 898:  DO[18181]=(OFF) ;
 899:  DO[834]=(ON) ;
 900:  DO[717]=(OFF) ;
 901:  !EZ1/SP1 schliessen ;
 902:  DO[718]=(ON) ;
 903:  !Fraeser ausblasen AUS/EIN ;
 904:  DO[847]=(F[330]) ;
 905:  TIMER[9]=((-4)) ;
 906:  !EZ1/SP1 Kraft erreicht ;
 907:  WAIT ((DI[718] AND !DI[772] AND !DI[780] AND !DI[774] AND !DI[775]) OR (TIMER[9]>=0))    ;
 908:  F[325]=((TIMER[9]>=0)) ;
 909:  DO[18181]=(ON) ;
 910:  DO[718]=((TIMER[9]<0)) ;
 911:  DO[834]=((TIMER[9]<0)) ;
 912:  WAIT ((DI[718] AND !DI[772] AND !DI[780] AND !DI[774] AND !DI[775]) OR DI[26] OR DI[27])    ;
 913:  DO[18181]=(OFF) ;
 914:  !EZ1/SP1 Fehler Kraftaufbau ;
 915:  IF (F[325]),JMP LBL[1201] ;
 916:  TIMER[9]=((-5)) ;
 917:  LBL[1200] ;
 918:  WAIT (!DI[834] OR F[325] OR (TIMER[9]>=0))    ;
 919:  WAIT (DI[834] OR F[325] OR (TIMER[9]>=0))    ;
 920:  R[1]=(R[1]+1) ;
 921:  F[329]=((TIMER[9]>=0)) ;
 922:  !Fraeszeit ueberschritten ;
 923:  IF (F[329]),JMP LBL[1201] ;
 924:  !Umdrehungen Vergleichen ;
 925:  IF (R[1]<R[4]),JMP LBL[1200] ;
 926:  !EZ1/SP1 2 Huebe bei NF ;
 927:  IF (!F[130]),JMP LBL[1201] ;
 928:  IF (F[98]),F[96]=(ON) ;
 929:  F[98]=(ON) ;
 930:  LBL[1201] ;
 931:  DO[834]=((TIMER[9]<0)) ;
 932:  !Fraeser ausblasen EIN ;
 933:  DO[847]=PULSE,4.0sec ;
 934:  !EZ1/SP1 oeffnen ;
 935:  DO[718]=(OFF) ;
 936:  DO[717]=(!DI[717]) ;
 937:  DO[18181]=(F[329]) ;
 938:  WAIT (!F[329] OR DI[26] OR DI[27])    ;
 939:  DO[18181]=(OFF) ;
 940:  DO[18181]=(ON) ;
 941:  WAIT (DI[717])    ;
 942:  DO[18181]=(OFF) ;
 943:  DO[717]=(OFF) ;
 944:  !Umdrehungen ruecksetzen ;
 945:  R[1]=0    ;
 946:  R[42]=12    ;
 947:  !Zähler umschreiben für 2ten Hub ;
 948:  IF (F[98] AND F[732]),GO[3]=36 ;
 949:  IF (F[96] AND F[732]),R[4]=R[45] ;
 950:  IF (F[329] OR F[325] OR (!F[96] AND F[130])),JMP LBL[12] ;
 951:  F[98]=(ON) ;
 952:  JMP LBL[13] ;
 953:   ;
 954:  !**************************** ;
 955:  !*        Schritt 13        * ;
 956:  !* STAT EZ1/SP1 i.O./n.i.O. * ;
 957:  !**************************** ;
 958:   ;
 959:  LBL[13] ;
 960:  R[41]=13    ;
 961:  !Fraesueberwachung starten ;
 962:  TIMER[7]=((-5)) ;
 963:  WAIT ((F[78] OR F[79]) AND (F[98] OR (F[94] AND F[96])) OR (TIMER[7]>=0))    ;
 964:  F[329]=((TIMER[7]>=0)) ;
 965:  IF (!F[329]),R[41]=14 ;
 966:  IF (F[329]),R[41]=12 ;
 967:  !KF1 U-Merker ruecksetzen ;
 968:  F[94]=(OFF) ;
 969:  F[96]=(OFF) ;
 970:  F[98]=(OFF) ;
 971:  R[42]=13    ;
 972:  JMP LBL[R[41]] ;
 973:   ;
 974:  !*************************** ;
 975:  !*       Schritt 14        * ;
 976:  !*    STAT EZ1/SP1 KS1     * ;
 977:  !* KS1 in Ruhest.schwenken * ;
 978:  !*************************** ;
 979:   ;
 980:  LBL[14] ;
 981:  R[41]=14    ;
 982:  !RSK gestartet ;
 983:  F[321]=(OFF) ;
 984:  DO[718]=(OFF) ;
 985:  DO[717]=(!DI[717]) ;
 986:  DO[18181]=(ON) ;
 987:  WAIT (DI[717])    ;
 988:  DO[18181]=(OFF) ;
 989:  DO[717]=(OFF) ;
 990:  TIMER[8]=((-4)) ;
 991:  WAIT ((DI[844] AND !DI[842] AND !DI[845] AND DI[843]) OR (TIMER[8]>=0))    ;
 992:  F[324]=((TIMER[8]>=0)) ;
 993:  DO[18181]=((TIMER[8]>=0)) ;
 994:  WAIT (DI[844] AND !DI[842] AND !DI[845] AND DI[843])    ;
 995:  DO[18181]=(OFF) ;
 996:  F[324]=(OFF) ;
 997:  TIMER[8]=((-4)) ;
 998:  DO[835]=(F[564]) ;
 999:  WAIT ((DI[835] AND F[564]) OR (!DI[835] AND !F[564]) OR (TIMER[8]>=0))    ;
1000:  F[323]=((TIMER[8]>=0)) ;
1001:  DO[18181]=((TIMER[8]>=0)) ;
1002:  WAIT ((DI[835] AND F[564]) OR (!DI[835] AND !F[564]))    ;
1003:  DO[18181]=(OFF) ;
1004:  F[323]=(OFF) ;
1005:  !Ueberwachungszeit KS1 Schwenken ;
1006:  TIMER[8]=((-4)) ;
1007:  DO[3969]=(ON) ;
1008:  WAIT (DI[841] OR (TIMER[8]>=0))    ;
1009:  DO[18181]=((TIMER[8]>=0)) ;
1010:  WAIT (DI[841])    ;
1011:  DO[18181]=(OFF) ;
1012:  TIMER[8]=((-6)) ;
1013:  WAIT ((!DI[844] AND DI[842] AND DI[845] AND !DI[843]) OR (TIMER[8]>=0))    ;
1014:  F[323]=((TIMER[8]>=0)) ;
1015:  DO[3969]=(OFF) ;
1016:  DO[18181]=((TIMER[8]>=0)) ;
1017:  WAIT ((!DI[844] AND DI[842] AND DI[845] AND !DI[843]) OR DI[26])    ;
1018:  DO[18181]=(OFF) ;
1019:  DO[835]=(OFF) ;
1020:  F[323]=(OFF) ;
1021:  DO[834]=(OFF) ;
1022:  !Sprung zurueck bei KS1 Fehler ;
1023:  IF (TIMER[8]>=0),JMP LBL[14] ;
1024:  R[42]=14    ;
1025:  JMP LBL[15] ;
1026:   ;
1027:  !*********************** ;
1028:  !*     Schritt 15      * ;
1029:  !*    STAT EZ1/SP1     * ;
1030:  !* Messen nach Fraesen * ;
1031:  !*********************** ;
1032:   ;
1033:  LBL[15] ;
1034:  R[41]=15    ;
1035:  !RSK gestartet ;
1036:  F[321]=(OFF) ;
1037:  GO[3]=1 ;
1038:  WAIT    .10(sec) ;
1039:  DO[786]=(ON) ;
1040:  DO[18181]=(ON) ;
1041:  WAIT (!DI[786] AND DI[787] AND !DI[788])    ;
1042:  DO[18181]=(OFF) ;
1043:  DO[786]=(OFF) ;
1044:  GO[1]=(31) ;
1045:  GO[3]=(31) ;
1046:  WAIT    .10(sec) ;
1047:  DO[757]=(ON) ;
1048:  TIMER[9]=((-8)) ;
1049:  WAIT (DI[757] OR (TIMER[9]>=0))    ;
1050:  F[326]=((TIMER[9]>=0)) ;
1051:  DO[18181]=(ON) ;
1052:  WAIT (DI[757] OR DI[26] OR DI[27])    ;
1053:  DO[18181]=(OFF) ;
1054:  F[326]=(OFF) ;
1055:  F[85]=(DI[776] OR DI[777]) ;
1056:  DO[757]=(OFF) ;
1057:  F[86]=(DI[736] OR (DI[735] AND DI[734] AND DI[733])) ;
1058:  TIMER[7]=((-2)) ;
1059:  WAIT ((!F[85] AND !F[86]) OR (TIMER[7]>=0))    ;
1060:  F[329]=((TIMER[7]>=0)) ;
1061:  DO[18181]=(F[329]) ;
1062:  WAIT ((!F[85] AND !F[86]) OR DI[26] OR DI[27])    ;
1063:  DO[18181]=(OFF) ;
1064:  F[329]=(OFF) ;
1065:  F[298]=(F[85] OR F[86]) ;
1066:  DO[717]=(!DI[717]) ;
1067:  DO[18181]=(ON) ;
1068:  WAIT ((DI[717] AND !DI[784]) OR (DI[717] AND F[298]))    ;
1069:  DO[18181]=(OFF) ;
1070:  DO[717]=(OFF) ;
1071:  R[42]=15    ;
1072:  !EZ1/SP1 wiederh. bei Messfehler ;
1073:  IF (DI[777]),JMP LBL[17] ;
1074:  DO[758]=(OFF) ;
1075:  DO[759]=(OFF) ;
1076:  !KS nicht bei K-Verschleiss ;
1077:  IF (F[298]),JMP LBL[9] ;
1078:  !EZ1/SP1 2.Setzhub nach Fraesen ;
1079:  IF (F[335] AND F[78]),JMP LBL[55] ;
1080:  !EZ1/SP1 Kurzschluss schweissen ;
1081:  IF (F[335] AND !F[78]),JMP LBL[16] ;
1082:  !EZ1/SP1 Kurzschluss schweissen ;
1083:  IF (!F[335]),JMP LBL[16] ;
1084:   ;
1085:  !************************** ;
1086:  !*       Schritt 16       * ;
1087:  !*      STAT EZ1/SP1      * ;
1088:  !* Kurzschlussschweissung * ;
1089:  !************************** ;
1090:   ;
1091:  LBL[16] ;
1092:  R[41]=16    ;
1093:  !RSK gestartet ;
1094:  F[321]=(OFF) ;
1095:  DO[145]=(ON) ;
1096:  !EZ1/SK1 Prog. ;
1097:  IF (F[78] AND !F[301]),GO[1]=(41) ;
1098:  IF (F[78] AND !F[301]),GO[3]=(41) ;
1099:  IF (F[79] OR F[301]),GO[1]=(51) ;
1100:  IF (F[79] OR F[301]),GO[3]=(51) ;
1101:  WAIT    .10(sec) ;
1102:  DO[717]=(OFF) ;
1103:  DO[718]=(OFF) ;
1104:  DO[785]=(OFF) ;
1105:  DO[514]=(OFF) ;
1106:  F[80]=(OFF) ;
1107:  F[306]=(OFF) ;
1108:  DO[18181]=(ON) ;
1109:  WAIT (DI[705] AND DI[713] AND DI[714] AND (!DI[784] OR (DI[769] AND DI[784])))    ;
1110:  DO[18181]=(OFF) ;
1111:  F[346]=(OFF) ;
1112:  DO[18181]=(ON) ;
1113:  WAIT ((!DI[785] AND DI[792] AND DI[802] AND !F[80]) OR (!DI[792] AND DI[802] AND DI[145]))    ;
1114:  DO[18181]=(OFF) ;
1115:  !EZ1/SP1 schliessen ;
1116:  DO[718]=(ON) ;
1117:  TIMER[9]=((-4)) ;
1118:  !EZ1/SP1 Kraft erreicht ;
1119:  WAIT ((DI[718] AND !DI[772] AND !DI[780]) OR DI[774] OR DI[775] OR (TIMER[9]>=0))    ;
1120:  DO[718]=(DI[718] AND !DI[774] AND !DI[775]) ;
1121:  DO[717]=(!DO[718]) ;
1122:  !Schweissen START ;
1123:  DO[785]=(DI[718] AND !DI[774] AND !DI[775]) ;
1124:  !EZ1/SP1 Fehler Ausgleich ;
1125:  F[302]=(DI[718] AND DI[719]) ;
1126:  !EZ1/SP1 Fehler SZ ;
1127:  F[300]=(DI[774] OR DI[775]) ;
1128:  !SK1 FK ;
1129:  TIMER[9]=((-1)) ;
1130:  WAIT ((F[80] AND DO[785]) OR ((DI[804] OR DI[805]) AND (DI[785] AND DO[785])) OR (DI[771] AND DI[784]) OR !DO[785] OR (TIMER[9]>=0))    ;
1131:  F[297]=(F[80] OR (DI[804] AND !DI[806] AND !DI[775] AND DI[785])) ;
1132:  !Fehler SK1 ;
1133:  F[301]=(!F[297] AND !F[298] AND DO[785]) ;
1134:  DO[785]=(OFF) ;
1135:  DO[718]=(OFF) ;
1136:  DO[18181]=(ON) ;
1137:  F[749]=(!F[297] AND !F[748]) ;
1138:  F[748]=(!F[297]) ;
1139:  WAIT (F[297] OR DI[26] OR DI[27] OR (F[749] AND F[731]))    ;
1140:  DO[910]=(OFF) ;
1141:  WAIT (!DI[26] AND !DI[27])    ;
1142:  DO[18181]=(OFF) ;
1143:  !EZ1/SP1 oeffnen ;
1144:  DO[717]=(!DI[717]) ;
1145:  TIMER[9]=((-4)) ;
1146:  WAIT (DI[717] OR (TIMER[9]>=0))    ;
1147:  F[303]=((TIMER[9]>=0)) ;
1148:  DO[18181]=(F[303]) ;
1149:  WAIT (DI[717])    ;
1150:  DO[18181]=(OFF) ;
1151:  F[303]=(OFF) ;
1152:  DO[717]=(OFF) ;
1153:  DO[145]=(OFF) ;
1154:  R[42]=16    ;
1155:  JMP LBL[17] ;
1156:   ;
1157:  !************************** ;
1158:  !*       Schritt 17       * ;
1159:  !*      STAT EZ1/SP1      * ;
1160:  !************************** ;
1161:   ;
1162:  LBL[17] ;
1163:  R[41]=17    ;
1164:  !RSK gestartet ;
1165:  F[321]=(OFF) ;
1166:  !Sprung zurueck bei Fehler ;
1167:  IF (!F[297] AND !DI[777]),JMP LBL[9] ;
1168:  !STAT EZ1/SP1 FK Fraesen ;
1169:  F[93]=(!F[329]) ;
1170:  DO[116]=(OFF) ;
1171:  DO[130]=(OFF) ;
1172:  R[42]=17    ;
1173:  JMP LBL[1] ;
1174:   ;
1175:   ;
1176:  !************************ ;
1177:  !************************ ;
1178:  !* Fraesen STAT EZ2/SP2 * ;
1179:  !************************ ;
1180:  !************************ ;
1181:   ;
1182:   ;
1183:  !****************************** ;
1184:  !*        Schritt 18          * ;
1185:  !*     STAT EZ2/SP2 KS2       * ;
1186:  !* KS2 in Arbeitsst.schwenken * ;
1187:  !****************************** ;
1188:   ;
1189:  LBL[18] ;
1190:  R[41]=18    ;
1191:  !RSK gestartet ;
1192:  F[321]=(OFF) ;
1193:  GO[4]=(31) ;
1194:  IF (F[285]),GO[3]=(35) ;
1195:  IF (!F[285]),GO[6]=(31) ;
1196:  WAIT    .10(sec) ;
1197:  DO[918]=(F[138]) ;
1198:  DO[919]=(F[139]) ;
1199:  DO[116]=(ON) ;
1200:  DO[162]=(ON) ;
1201:  DO[878]=(OFF) ;
1202:  DO[877]=(!DI[877]) ;
1203:  DO[18181]=(ON) ;
1204:  WAIT (DI[877])    ;
1205:  DO[18181]=(OFF) ;
1206:  DO[877]=(OFF) ;
1207:  !Ueberwachungszeit Grundstellung ;
1208:  TIMER[8]=((-4)) ;
1209:  WAIT ((!DI[1004] AND DI[1002] AND DI[1005] AND !DI[1003]) OR (TIMER[8]>=0))    ;
1210:  F[323]=((TIMER[8]>=0)) ;
1211:  DO[18181]=((TIMER[8]>=0)) ;
1212:  WAIT (!DI[1004] AND DI[1002] AND DI[1005] AND !DI[1003])    ;
1213:  DO[18181]=(OFF) ;
1214:  F[323]=(OFF) ;
1215:  TIMER[8]=((-4)) ;
1216:  DO[995]=(F[564]) ;
1217:  WAIT ((DI[995] AND F[564]) OR (!DI[995] AND !F[564]) OR (TIMER[8]>=0))    ;
1218:  F[323]=((TIMER[8]>=0)) ;
1219:  DO[18181]=((TIMER[8]>=0)) ;
1220:  WAIT ((DI[995] AND F[564]) OR (!DI[995] AND !F[564]))    ;
1221:  DO[18181]=(OFF) ;
1222:  F[323]=(OFF) ;
1223:  !Ueberwachungszeit KS2 Schwenken ;
1224:  TIMER[8]=((-6)) ;
1225:  DO[3973]=(ON) ;
1226:  DO[18181]=(ON) ;
1227:  WAIT (DI[1001])    ;
1228:  DO[18181]=(OFF) ;
1229:  WAIT ((DI[1004] AND !DI[1002] AND !DI[1005] AND DI[1003]) OR (TIMER[8]>=0))    ;
1230:  F[324]=((TIMER[8]>=0)) ;
1231:  DO[3973]=(OFF) ;
1232:  DO[18181]=((TIMER[8]>=0)) ;
1233:  WAIT ((DI[1004] AND !DI[1002] AND !DI[1005] AND DI[1003]) OR DI[26])    ;
1234:  DO[18181]=(OFF) ;
1235:  F[324]=(OFF) ;
1236:  !Sprung zurueck bei KS2 Fehler ;
1237:  IF (TIMER[8]>=0),JMP LBL[18] ;
1238:  DO[995]=(OFF) ;
1239:  TIMER[11]=((R[24])) ;
1240:  WAIT ((TIMER[11]>=0) OR !F[564])    ;
1241:  TIMER[11]=STOP ;
1242:  DO[18181]=(ON) ;
1243:  WAIT ((F[148] AND F[138]) OR (F[148] AND F[139]))    ;
1244:  DO[18181]=(OFF) ;
1245:  !Anwahl Startfraesen ;
1246:  IF (!DI[1002] AND DI[1003] AND F[148] AND F[138] AND !F[301]),R[41]=19 ;
1247:  !Anwahl Normalfraesen ;
1248:  IF (!DI[1002] AND DI[1003] AND F[148] AND (F[139] OR F[301])),R[41]=21 ;
1249:  R[42]=18    ;
1250:  JMP LBL[R[41]] ;
1251:   ;
1252:  !************************** ;
1253:  !*      Schritt 19        * ;
1254:  !* STAT EZ2/SP2 SF Teil 1 * ;
1255:  !************************** ;
1256:   ;
1257:  LBL[19] ;
1258:  R[41]=19    ;
1259:  !RSK gestartet ;
1260:  F[321]=(OFF) ;
1261:  F[329]=(OFF) ;
1262:  F[325]=(OFF) ;
1263:  DO[878]=(OFF) ;
1264:  DO[877]=(!DI[877]) ;
1265:  DO[18181]=(ON) ;
1266:  WAIT (DI[877])    ;
1267:  DO[18181]=(OFF) ;
1268:  DO[994]=(ON) ;
1269:  DO[877]=(OFF) ;
1270:  !Warte Fraeser laeuft ;
1271:  TIMER[7]=((-3)) ;
1272:  WAIT (!DI[994] OR (TIMER[7]>=0))    ;
1273:  WAIT (DI[994] OR (TIMER[7]>=0))    ;
1274:  F[322]=((TIMER[7]>=0)) ;
1275:  DO[18181]=(ON) ;
1276:  WAIT (!DI[994])    ;
1277:  WAIT (DI[994])    ;
1278:  DO[18181]=(OFF) ;
1279:  F[322]=(OFF) ;
1280:  !EZ2/SP2 schliessen ;
1281:  DO[878]=(ON) ;
1282:  !Fraeser ausblasen AUS/EIN ;
1283:  DO[1007]=(F[330]) ;
1284:  TIMER[9]=((-4)) ;
1285:  !EZ2/SP2 Kraft erreicht ;
1286:  WAIT ((DI[878] AND !DI[932] AND !DI[940] AND !DI[934] AND !DI[935]) OR (TIMER[9]>=0))    ;
1287:  F[325]=((TIMER[9]>=0)) ;
1288:  DO[18181]=(ON) ;
1289:  DO[878]=((TIMER[9]<0)) ;
1290:  DO[994]=((TIMER[9]<0)) ;
1291:  WAIT ((DI[878] AND !DI[932] AND !DI[940] AND !DI[934] AND !DI[935]) OR DI[26] OR DI[27])    ;
1292:  DO[18181]=(OFF) ;
1293:  F[325]=(OFF) ;
1294:  !EZ2/SP2 Fehler Kraftaufbau ;
1295:  IF (F[325]),JMP LBL[1901] ;
1296:  TIMER[9]=((-5)) ;
1297:  LBL[1900] ;
1298:  WAIT (!DI[994] OR F[325] OR (TIMER[9]>=0))    ;
1299:  WAIT (DI[994] OR F[325] OR (TIMER[9]>=0))    ;
1300:  R[1]=(R[1]+1) ;
1301:  F[329]=((TIMER[9]>=0)) ;
1302:  !Fraeszeit ueberschritten ;
1303:  IF (F[329]),JMP LBL[1901] ;
1304:  !Umdrehungen Vergleichen ;
1305:  IF (R[1]<R[5]),JMP LBL[1900] ;
1306:  F[150]=(ON) ;
1307:  LBL[1901] ;
1308:  DO[994]=((TIMER[9]<0)) ;
1309:  !Fraeser ausblasen EIN ;
1310:  DO[1007]=(F[330] OR (TIMER[9]<0)) ;
1311:  DO[878]=(OFF) ;
1312:  !EZ2/SP2 oeffnen ;
1313:  DO[877]=(!DI[877]) ;
1314:  DO[18181]=(F[329]) ;
1315:  WAIT (!F[329] OR DI[26] OR DI[27])    ;
1316:  DO[18181]=(OFF) ;
1317:  DO[18181]=(ON) ;
1318:  WAIT (DI[877])    ;
1319:  DO[18181]=(OFF) ;
1320:  DO[877]=(OFF) ;
1321:  !Umdrehungen ruecksetzen ;
1322:  R[1]=0    ;
1323:  R[42]=19    ;
1324:  IF (F[329] OR F[325]),JMP LBL[19] ;
1325:  JMP LBL[20] ;
1326:   ;
1327:  !************************** ;
1328:  !*       Schritt 20       * ;
1329:  !* STAT EZ2/SP2 SF Teil 2 * ;
1330:  !************************** ;
1331:   ;
1332:  LBL[20] ;
1333:  R[41]=20    ;
1334:  !RSK gestartet ;
1335:  F[321]=(OFF) ;
1336:  F[329]=(OFF) ;
1337:  F[325]=(OFF) ;
1338:  DO[878]=(OFF) ;
1339:  DO[877]=(!DI[877]) ;
1340:  DO[18181]=(ON) ;
1341:  WAIT (DI[877])    ;
1342:  DO[18181]=(OFF) ;
1343:  DO[994]=(ON) ;
1344:  DO[877]=(OFF) ;
1345:  !Zange zu... ;
1346:  DO[878]=(ON) ;
1347:  !Fraeser ausblasen AUS/EIN ;
1348:  DO[1007]=(F[330]) ;
1349:  TIMER[9]=((-4)) ;
1350:  !EZ2/SP2 Kraft erreicht ;
1351:  WAIT ((DI[878] AND !DI[932] AND !DI[940] AND !DI[934] AND !DI[935]) OR (TIMER[9]>=0))    ;
1352:  F[325]=((TIMER[9]>=0)) ;
1353:  DO[18181]=(ON) ;
1354:  DO[878]=((TIMER[9]<0)) ;
1355:  DO[994]=((TIMER[9]<0)) ;
1356:  WAIT ((DI[878] AND !DI[932] AND !DI[940] AND !DI[934] AND !DI[935]) OR DI[26] OR DI[27])    ;
1357:  DO[18181]=(OFF) ;
1358:  !EZ2/SP2 Fehler Kraftaufbau ;
1359:  IF (F[325]),JMP LBL[2001] ;
1360:  TIMER[9]=((-5)) ;
1361:  LBL[2000] ;
1362:  WAIT (!DI[994] OR F[325] OR (TIMER[9]>=0))    ;
1363:  WAIT (DI[994] OR F[325] OR (TIMER[9]>=0))    ;
1364:  R[1]=(R[1]+1) ;
1365:  F[329]=((TIMER[9]>=0)) ;
1366:  !Fraeszeit ueberschritten ;
1367:  IF (F[329]),JMP LBL[2001] ;
1368:  !Umdrehungen Vergleichen ;
1369:  IF (R[1]<R[6]),JMP LBL[2000] ;
1370:  F[152]=(ON) ;
1371:  LBL[2001] ;
1372:  DO[994]=((TIMER[9]<0)) ;
1373:  !Fraeser ausblasen EIN ;
1374:  DO[1007]=PULSE,4.0sec ;
1375:  DO[878]=(OFF) ;
1376:  !EZ2/SP2 oeffnen ;
1377:  DO[877]=(!DI[877]) ;
1378:  DO[18181]=(F[329]) ;
1379:  WAIT (!F[329] OR DI[26] OR DI[27])    ;
1380:  DO[18181]=(OFF) ;
1381:  DO[18181]=(ON) ;
1382:  WAIT (DI[877])    ;
1383:  DO[18181]=(OFF) ;
1384:  DO[877]=(OFF) ;
1385:  !Umdrehungen ruecksetzen ;
1386:  R[1]=0    ;
1387:  R[42]=20    ;
1388:  IF (F[329] OR F[325]),JMP LBL[20] ;
1389:  JMP LBL[22] ;
1390:   ;
1391:  !********************* ;
1392:  !*     Schritt 21    * ;
1393:  !*   STAT EZ2/SP2 NF * ;
1394:  !********************* ;
1395:   ;
1396:  LBL[21] ;
1397:  R[41]=21    ;
1398:  !RSK gestartet ;
1399:  F[321]=(OFF) ;
1400:  F[329]=(OFF) ;
1401:  F[325]=(OFF) ;
1402:  !Zähler wegspeichern für 2ten Hub ;
1403:  R[45]=R[7]    ;
1404:  IF (F[154] AND F[732]),R[7]=R[44] ;
1405:  DO[878]=(OFF) ;
1406:  DO[877]=(!DI[877]) ;
1407:  DO[18181]=(ON) ;
1408:  WAIT (DI[877])    ;
1409:  DO[18181]=(OFF) ;
1410:  DO[994]=(ON) ;
1411:  DO[877]=(OFF) ;
1412:  !EZ2/SP2 schliessen ;
1413:  DO[878]=(ON) ;
1414:  !Fraeser ausblasen AUS ;
1415:  DO[1007]=(F[330]) ;
1416:  TIMER[9]=((-4)) ;
1417:  !EZ2/SP2 Kraft erreicht ;
1418:  WAIT ((DI[878] AND !DI[932] AND !DI[940] AND !DI[934] AND !DI[935]) OR (TIMER[9]>=0))    ;
1419:  F[325]=((TIMER[9]>=0)) ;
1420:  DO[18181]=(ON) ;
1421:  DO[878]=((TIMER[9]<0)) ;
1422:  DO[994]=((TIMER[9]<0)) ;
1423:  WAIT ((DI[878] AND !DI[932] AND !DI[940] AND !DI[934] AND !DI[935]) OR DI[26] OR DI[27])    ;
1424:  DO[18181]=(OFF) ;
1425:  !EZ2/SP2 Fehler Kraftaufbau ;
1426:  IF (F[325]),JMP LBL[2101] ;
1427:  TIMER[9]=((-5)) ;
1428:  LBL[2100] ;
1429:  WAIT (!DI[994] OR F[325] OR (TIMER[9]>=0))    ;
1430:  WAIT (DI[994] OR F[325] OR (TIMER[9]>=0))    ;
1431:  R[1]=(R[1]+1) ;
1432:  F[329]=((TIMER[9]>=0)) ;
1433:  !Fraeszeit ueberschritten ;
1434:  IF (F[329]),JMP LBL[2101] ;
1435:  !Umdrehungen Vergleichen ;
1436:  IF (R[1]<R[7]),JMP LBL[2100] ;
1437:  !EZ2/SP2 2 Huebe bei NF ;
1438:  IF (!F[164]),JMP LBL[2101] ;
1439:  IF (F[154]),F[152]=(ON) ;
1440:  F[154]=(ON) ;
1441:  LBL[2101] ;
1442:  DO[878]=(OFF) ;
1443:  DO[994]=((TIMER[9]<0)) ;
1444:  !Fraeser ausblasen EIN ;
1445:  DO[1007]=PULSE,4.0sec ;
1446:  !EZ2/SP2 oeffnen ;
1447:  DO[877]=(!DI[877]) ;
1448:  DO[18181]=(F[329]) ;
1449:  WAIT (!F[329] OR DI[26] OR DI[27])    ;
1450:  DO[18181]=(OFF) ;
1451:  DO[18181]=(ON) ;
1452:  WAIT (DI[877])    ;
1453:  DO[18181]=(OFF) ;
1454:  DO[877]=(OFF) ;
1455:  !Umdrehungen ruecksetzen ;
1456:  R[1]=0    ;
1457:  R[42]=21    ;
1458:  !Zähler umschreiben für 2ten Hub ;
1459:  IF (F[154] AND F[732]),GO[3]=36 ;
1460:  IF (F[152] AND F[732]),R[7]=R[45] ;
1461:  IF (F[329] OR F[325] OR (!F[152] AND F[164])),JMP LBL[21] ;
1462:  F[154]=(ON) ;
1463:  JMP LBL[22] ;
1464:   ;
1465:  !*************************** ;
1466:  !*        Schritt 22       * ;
1467:  !* STAT EZ2/SP2 i.O/n.i.O. * ;
1468:  !*************************** ;
1469:   ;
1470:  LBL[22] ;
1471:  R[41]=22    ;
1472:  !Fraesueberwachung starten ;
1473:  TIMER[7]=((-5)) ;
1474:  WAIT ((F[138] OR F[139]) AND (F[154] OR (F[150] AND F[152])) OR (TIMER[7]>=0))    ;
1475:  F[329]=((TIMER[7]>=0)) ;
1476:  IF (!F[329]),R[41]=23 ;
1477:  IF (F[329]),R[41]=21 ;
1478:  !KF1 U-Merker ruecksetzen ;
1479:  F[150]=(OFF) ;
1480:  F[152]=(OFF) ;
1481:  F[154]=(OFF) ;
1482:  R[42]=22    ;
1483:  JMP LBL[R[41]] ;
1484:   ;
1485:  !*************************** ;
1486:  !*       Schritt 23        * ;
1487:  !*      STAT EZ2/SP2       * ;
1488:  !* KS2 in Ruhest.schwenken * ;
1489:  !*************************** ;
1490:   ;
1491:  LBL[23] ;
1492:  R[41]=23    ;
1493:  !RSK gestartet ;
1494:  F[321]=(OFF) ;
1495:  DO[878]=(OFF) ;
1496:  DO[877]=(!DI[877]) ;
1497:  DO[18181]=(ON) ;
1498:  WAIT (DI[877])    ;
1499:  DO[18181]=(OFF) ;
1500:  DO[877]=(OFF) ;
1501:  TIMER[8]=((-4)) ;
1502:  WAIT ((DI[1004] AND !DI[1002] AND !DI[1005] AND DI[1003]) OR (TIMER[8]>=0))    ;
1503:  F[324]=((TIMER[8]>=0)) ;
1504:  DO[18181]=((TIMER[8]>=0)) ;
1505:  WAIT (DI[1004] AND !DI[1002] AND !DI[1005] AND DI[1003])    ;
1506:  DO[18181]=(OFF) ;
1507:  F[324]=(OFF) ;
1508:  TIMER[8]=((-4)) ;
1509:  DO[995]=(F[564]) ;
1510:  WAIT ((DI[995] AND F[564]) OR (!DI[995] AND !F[564]) OR (TIMER[8]>=0))    ;
1511:  F[323]=((TIMER[8]>=0)) ;
1512:  DO[18181]=((TIMER[8]>=0)) ;
1513:  WAIT ((DI[995] AND F[564]) OR (!DI[995] AND !F[564]))    ;
1514:  DO[18181]=(OFF) ;
1515:  F[323]=(OFF) ;
1516:  !Ueberwachungszeit KS2 Schwenken ;
1517:  TIMER[8]=((-4)) ;
1518:  DO[3970]=(ON) ;
1519:  WAIT (DI[1001] OR (TIMER[8]>=0))    ;
1520:  DO[18181]=((TIMER[8]>=0)) ;
1521:  WAIT (DI[1001])    ;
1522:  TIMER[8]=((-6)) ;
1523:  DO[18181]=(OFF) ;
1524:  WAIT ((!DI[1004] AND DI[1002] AND DI[1005] AND !DI[1003]) OR (TIMER[8]>=0))    ;
1525:  F[323]=((TIMER[8]>=0)) ;
1526:  DO[3970]=(OFF) ;
1527:  DO[18181]=((TIMER[8]>=0)) ;
1528:  WAIT ((!DI[1004] AND DI[1002] AND DI[1005] AND !DI[1003]) OR DI[26])    ;
1529:  DO[18181]=(OFF) ;
1530:  F[323]=(OFF) ;
1531:  DO[995]=(OFF) ;
1532:  DO[994]=(OFF) ;
1533:  !Sprung zurueck bei KS2 Fehler ;
1534:  IF (TIMER[8]>=0),JMP LBL[23] ;
1535:  R[42]=23    ;
1536:  JMP LBL[24] ;
1537:   ;
1538:  !*********************** ;
1539:  !*     Schritt 24      * ;
1540:  !*    STAT EZ2/SP2     * ;
1541:  !* Messen nach Fraesen * ;
1542:  !*********************** ;
1543:   ;
1544:  LBL[24] ;
1545:  R[41]=24    ;
1546:  !RSK gestartet ;
1547:  F[321]=(OFF) ;
1548:  IF (!F[285]),JMP LBL[2400] ;
1549:  IF (F[285]),JMP LBL[2401] ;
1550:  LBL[2400] ;
1551:  GO[6]=1 ;
1552:  WAIT    .10(sec) ;
1553:  DO[946]=(ON) ;
1554:  !STAT EZ2/SP2 FK Fraesen ;
1555:  DO[18181]=(ON) ;
1556:  WAIT (!DI[946] AND DI[947] AND !DI[948])    ;
1557:  DO[18181]=(OFF) ;
1558:  DO[946]=(OFF) ;
1559:  JMP LBL[2402] ;
1560:  LBL[2401] ;
1561:  IF (!F[285]),GO[3]=(1) ;
1562:  IF (F[285]),GO[3]=(5) ;
1563:  WAIT    .10(sec) ;
1564:  DO[786]=(ON) ;
1565:  !STAT EZ2/SP2 FK Fraesen ;
1566:  DO[18181]=(ON) ;
1567:  WAIT (!DI[786] AND DI[787] AND !DI[788])    ;
1568:  DO[18181]=(OFF) ;
1569:  DO[786]=(OFF) ;
1570:  LBL[2402] ;
1571:  GO[4]=(31) ;
1572:  IF (F[285]),GO[3]=(35) ;
1573:  IF (!F[285]),GO[6]=(31) ;
1574:  WAIT    .10(sec) ;
1575:  DO[917]=(ON) ;
1576:  TIMER[9]=((-8)) ;
1577:  WAIT (DI[917] OR (TIMER[9]>=0))    ;
1578:  F[326]=((TIMER[9]>=0)) ;
1579:  DO[18181]=(F[326]) ;
1580:  WAIT (DI[917] OR DI[26] OR DI[27])    ;
1581:  DO[18181]=(OFF) ;
1582:  F[326]=(OFF) ;
1583:  F[143]=(DI[936] OR DI[937]) ;
1584:  DO[917]=(OFF) ;
1585:  F[144]=(DI[896] OR (DI[895] AND DI[894] AND DI[893])) ;
1586:  TIMER[7]=((-2)) ;
1587:  WAIT ((!F[144] AND !F[143]) OR (TIMER[7]>=0))    ;
1588:  F[329]=((TIMER[7]>=0)) ;
1589:  DO[18181]=(F[329]) ;
1590:  WAIT ((!F[144] AND !F[143]) OR DI[26] OR DI[27])    ;
1591:  DO[18181]=(OFF) ;
1592:  F[329]=(OFF) ;
1593:  F[298]=(F[144] OR F[143]) ;
1594:  DO[877]=(!DI[877]) ;
1595:  DO[18181]=(ON) ;
1596:  WAIT ((DI[877] AND !DI[944]) OR (DI[877] AND F[298]))    ;
1597:  DO[18181]=(OFF) ;
1598:  DO[877]=(OFF) ;
1599:  R[42]=24    ;
1600:  !EZ2/SP2 wiederh. bei Messfehler ;
1601:  IF (F[298]),JMP LBL[18] ;
1602:  DO[918]=(OFF) ;
1603:  DO[919]=(OFF) ;
1604:  !KS nicht bei K-Verschleiss ;
1605:  IF (DI[937]),JMP LBL[26] ;
1606:  !EZ2/SP2 2.Setzhub nach Fraesen ;
1607:  IF (F[335] AND F[138]),JMP LBL[56] ;
1608:  !EZ2/SP2 Kurzschluss schweissen ;
1609:  IF (F[335] AND !F[138]),JMP LBL[25] ;
1610:  !EZ2/SP2 Kurzschluss schweissen ;
1611:  IF (!F[335]),JMP LBL[25] ;
1612:   ;
1613:  !************************** ;
1614:  !*       Schritt 25       * ;
1615:  !*      STAT EZ2/SP2      * ;
1616:  !* Kurzschlussschweissung * ;
1617:  !************************** ;
1618:   ;
1619:  LBL[25] ;
1620:  R[41]=25    ;
1621:  !RSK gestartet ;
1622:  F[321]=(OFF) ;
1623:  DO[145]=(F[285]) ;
1624:  DO[177]=(!F[285]) ;
1625:  !EZ2/SP2 SK1/SK2 Prog. ;
1626:  IF (F[285] AND F[138] AND !F[301]),GO[3]=(45) ;
1627:  IF (!F[285] AND F[138] AND !F[301]),GO[4]=(41) ;
1628:  IF (!F[285] AND F[138] AND !F[301]),GO[6]=(41) ;
1629:  IF ((F[285] AND F[139]) OR (F[285] AND F[301])),GO[3]=(55) ;
1630:  IF ((!F[285] AND F[139]) OR (!F[285] AND F[301])),GO[4]=(51) ;
1631:  IF ((!F[285] AND F[139]) OR (!F[285] AND F[301])),GO[6]=(51) ;
1632:  WAIT    .10(sec) ;
1633:  DO[877]=(OFF) ;
1634:  DO[878]=(OFF) ;
1635:  DO[945]=(OFF) ;
1636:  DO[785]=(!F[285] AND DO[785]) ;
1637:  DO[514]=(ON) ;
1638:  F[140]=(OFF) ;
1639:  F[80]=(OFF) ;
1640:  F[142]=(!F[285]) ;
1641:  F[306]=(OFF) ;
1642:  F[303]=(!DI[929] AND DI[944]) ;
1643:  DO[18181]=(ON) ;
1644:  WAIT (DI[865] AND DI[873] AND DI[874] AND (!DI[944] OR (DI[929] AND DI[944])))    ;
1645:  F[303]=(OFF) ;
1646:  WAIT ((!DI[945] AND DI[952] AND DI[962] AND !F[140]) OR (!DI[952] AND DI[962] AND !DI[913]) OR F[285])    ;
1647:  WAIT ((!DI[785] AND DI[792] AND DI[802] AND !F[80]) OR (!DI[792] AND DI[802] AND !DI[913]) OR !F[285])    ;
1648:  DO[18181]=(OFF) ;
1649:  !EZ2/SP2 schliessen ;
1650:  DO[878]=(ON) ;
1651:  TIMER[9]=((-4)) ;
1652:  WAIT ((DI[878] AND !DI[932] AND !DI[940]) OR DI[934] OR DI[935] OR (TIMER[9]>=0))    ;
1653:  DO[878]=(DI[878] AND !DI[934] AND !DI[935]) ;
1654:  DO[877]=(!DO[878]) ;
1655:  !Schweissen START ;
1656:  DO[945]=(DI[878] AND !DI[934] AND !DI[935] AND !F[285]) ;
1657:  DO[785]=((DI[878] AND !DI[934] AND !DI[935] AND F[285]) OR (!F[285] AND DO[785])) ;
1658:  !EZ2/SP2 Fehler Ausgleich ;
1659:  F[302]=(DI[878] AND DI[879]) ;
1660:  !EZ2/SP2 Fehler SZ ;
1661:  F[300]=(DI[934] OR DI[935]) ;
1662:  !SK1/SK2 FK ;
1663:  TIMER[9]=((-10)) ;
1664:  WAIT ((F[140] AND DO[945]) OR ((DI[964] OR DI[965]) AND (DI[945] AND DO[945])) OR (DI[931] AND DI[944]) OR (!DO[945] AND F[285]) OR (TIMER[9]>=0))    ;
1665:  WAIT ((F[80] AND DO[785]) OR ((DI[804] OR DI[805]) AND (DI[785] AND DO[785])) OR (DI[931] AND DI[944]) OR (!DO[785] AND !F[285]) OR (TIMER[9]>=0))    ;
1666:  F[297]=(F[140] OR (!DI[935] AND DI[945] AND DI[964] AND !DI[966]) OR F[80] OR (!DI[935] AND DI[785] AND DI[804] AND !DI[806])) ;
1667:  !Fehler SK1/SK2 ;
1668:  F[301]=(!F[297] AND !F[298] AND (DO[785] OR DO[945])) ;
1669:  DO[945]=(OFF) ;
1670:  DO[878]=(OFF) ;
1671:  DO[785]=((F[285] AND !DI[785]) OR (!F[285] AND DO[785])) ;
1672:  F[327]=(!F[297]) ;
1673:  DO[18181]=(F[327]) ;
1674:  F[749]=(!F[297] AND !F[748]) ;
1675:  F[748]=(!F[297]) ;
1676:  WAIT (F[297] OR DI[26] OR DI[27] OR (F[749] AND F[731]))    ;
1677:  F[327]=(OFF) ;
1678:  WAIT (!DI[26] AND !DI[27])    ;
1679:  DO[18181]=(OFF) ;
1680:  !EZ2/SP2 oeffnen ;
1681:  DO[877]=(!DI[877]) ;
1682:  TIMER[9]=((-4)) ;
1683:  WAIT (DI[877] OR (TIMER[9]>=0))    ;
1684:  F[303]=((TIMER[9]>=0)) ;
1685:  DO[18181]=(F[303]) ;
1686:  WAIT (DI[877])    ;
1687:  DO[18181]=(OFF) ;
1688:  F[303]=(OFF) ;
1689:  DO[877]=(OFF) ;
1690:  DO[145]=(OFF) ;
1691:  DO[177]=(OFF) ;
1692:  R[42]=25    ;
1693:  JMP LBL[26] ;
1694:   ;
1695:  !****************************** ;
1696:  !*         Schritt 26         * ;
1697:  !*       STAT EZ2/SP2 FK      * ;
1698:  !****************************** ;
1699:   ;
1700:  LBL[26] ;
1701:  R[41]=26    ;
1702:  !RSK gestartet ;
1703:  F[321]=(OFF) ;
1704:  !Sprung zurueck bei Fehler ;
1705:  IF (!F[297] AND !DI[937]),JMP LBL[18] ;
1706:  !STAT EZ2/SP2 FK Fraesen ;
1707:  F[149]=(!F[329]) ;
1708:  DO[116]=(OFF) ;
1709:  DO[162]=(OFF) ;
1710:  R[42]=26    ;
1711:  JMP LBL[1] ;
1712:   ;
1713:   ;
1714:  !************************ ;
1715:  !************************ ;
1716:  !* Fraesen STAT EZ3/SP3 * ;
1717:  !************************ ;
1718:  !************************ ;
1719:   ;
1720:   ;
1721:  !******************************* ;
1722:  !*        Schritt 27           * ;
1723:  !*       STAT EZ3/SP3          * ;
1724:  !* KS3 in Arbeitsst. schwenken * ;
1725:  !******************************* ;
1726:   ;
1727:  LBL[27] ;
1728:  R[41]=27    ;
1729:  !RSK gestartet ;
1730:  F[321]=(OFF) ;
1731:  GO[7]=(31) ;
1732:  GO[9]=(31) ;
1733:  WAIT    .10(sec) ;
1734:  DO[1078]=(F[174]) ;
1735:  DO[1079]=(F[175]) ;
1736:  DO[116]=(ON) ;
1737:  DO[194]=(ON) ;
1738:  DO[1038]=(OFF) ;
1739:  DO[1037]=(!DI[1037]) ;
1740:  DO[18181]=(ON) ;
1741:  WAIT (DI[1037])    ;
1742:  DO[18181]=(OFF) ;
1743:  DO[1037]=(OFF) ;
1744:  !Ueberwachungszeit Grundstellung ;
1745:  TIMER[8]=((-4)) ;
1746:  WAIT ((DI[1162] AND !DI[1163] AND !DI[1164] AND DI[1165]) OR (TIMER[8]>=0))    ;
1747:  F[323]=((TIMER[8]>=0)) ;
1748:  DO[18181]=((TIMER[8]>=0)) ;
1749:  WAIT (DI[1162] AND !DI[1163] AND !DI[1164] AND DI[1165])    ;
1750:  DO[18181]=(OFF) ;
1751:  F[323]=(OFF) ;
1752:  TIMER[8]=((-4)) ;
1753:  DO[1155]=(F[564]) ;
1754:  WAIT ((DI[1155] AND F[564]) OR (!DI[1155] AND !F[564]) OR (TIMER[8]>=0))    ;
1755:  F[323]=((TIMER[8]>=0)) ;
1756:  DO[18181]=((TIMER[8]>=0)) ;
1757:  WAIT ((DI[1155] AND F[564]) OR (!DI[1155] AND !F[564]))    ;
1758:  DO[18181]=(OFF) ;
1759:  F[323]=(OFF) ;
1760:  !Ueberwachungszeit KS3 Schwenken ;
1761:  TIMER[8]=((-4)) ;
1762:  DO[3974]=(ON) ;
1763:  WAIT (DI[1161] OR (TIMER[8]>=0))    ;
1764:  DO[18181]=((TIMER[8]>=0)) ;
1765:  WAIT (DI[1161])    ;
1766:  TIMER[8]=((-6)) ;
1767:  DO[18181]=(OFF) ;
1768:  WAIT ((!DI[1162] AND DI[1163] AND DI[1164] AND !DI[1165]) OR (TIMER[8]>=0))    ;
1769:  F[324]=((TIMER[8]>=0)) ;
1770:  DO[3974]=(OFF) ;
1771:  DO[18181]=((TIMER[8]>=0)) ;
1772:  WAIT ((!DI[1162] AND DI[1163] AND DI[1164] AND !DI[1165]) OR DI[26])    ;
1773:  DO[18181]=(OFF) ;
1774:  F[324]=(OFF) ;
1775:  !Sprung zurueck bei KS3 Fehler ;
1776:  IF (TIMER[8]>=0),JMP LBL[27] ;
1777:  DO[1155]=(OFF) ;
1778:  TIMER[11]=((R[24])) ;
1779:  WAIT ((TIMER[11]>=0) OR !F[564])    ;
1780:  TIMER[11]=STOP ;
1781:  DO[18181]=(ON) ;
1782:  WAIT ((F[184] AND F[174]) OR (F[184] AND F[175]))    ;
1783:  DO[18181]=(OFF) ;
1784:  !Anwahl Startfraesen ;
1785:  IF (!DI[1162] AND DI[1163] AND F[184] AND F[174] AND !F[301]),R[41]=28 ;
1786:  !Anwahl Normalfraesen ;
1787:  IF (!DI[1162] AND DI[1163] AND F[184] AND (F[175] OR F[301])),R[41]=30 ;
1788:  R[42]=27    ;
1789:  JMP LBL[R[41]] ;
1790:   ;
1791:  !************************** ;
1792:  !*       Schritt 28       * ;
1793:  !* STAT EZ3/SP3 SF Teil 1 * ;
1794:  !************************** ;
1795:   ;
1796:  LBL[28] ;
1797:  R[41]=28    ;
1798:  !RSK gestartet ;
1799:  F[321]=(OFF) ;
1800:  F[329]=(OFF) ;
1801:  F[325]=(OFF) ;
1802:  DO[1038]=(OFF) ;
1803:  DO[1037]=(!DI[1037]) ;
1804:  DO[18181]=(ON) ;
1805:  WAIT (DI[1037])    ;
1806:  DO[1037]=(OFF) ;
1807:  DO[18181]=(OFF) ;
1808:  DO[1154]=(ON) ;
1809:  !Warte Fraeser laeuft ;
1810:  TIMER[7]=((-3)) ;
1811:  WAIT (!DI[1154] OR (TIMER[7]>=0))    ;
1812:  WAIT (DI[1154] OR (TIMER[7]>=0))    ;
1813:  F[322]=((TIMER[7]>=0)) ;
1814:  DO[18181]=(ON) ;
1815:  WAIT (!DI[1154])    ;
1816:  WAIT (DI[1154])    ;
1817:  DO[18181]=(OFF) ;
1818:  F[322]=(OFF) ;
1819:  !EZ3/SP3 schliessen ;
1820:  DO[1038]=(ON) ;
1821:  !Fraeser ausblasen AUS/EIN ;
1822:  DO[1167]=(F[330]) ;
1823:  TIMER[9]=((-4)) ;
1824:  !EZ3/SP3 Kraft erreicht ;
1825:  WAIT ((DI[1038] AND !DI[1092] AND !DI[1100] AND !DI[1094] AND !DI[1095]) OR (TIMER[9]>=0))    ;
1826:  F[325]=((TIMER[9]>=0)) ;
1827:  DO[18181]=(ON) ;
1828:  DO[1038]=((TIMER[9]<0)) ;
1829:  DO[1154]=((TIMER[9]<0)) ;
1830:  WAIT ((DI[1038] AND !DI[1092] AND !DI[1100] AND !DI[1094] AND !DI[1095]) OR DI[26] OR DI[27])    ;
1831:  DO[18181]=(OFF) ;
1832:  !EZ3/SP3 Fehler Kraftaufbau ;
1833:  IF (F[325]),JMP LBL[2801] ;
1834:  TIMER[9]=((-5)) ;
1835:  LBL[2800] ;
1836:  WAIT (!DI[1154] OR F[325] OR (TIMER[9]>=0))    ;
1837:  WAIT (DI[1154] OR F[325] OR (TIMER[9]>=0))    ;
1838:  R[1]=(R[1]+1) ;
1839:  F[329]=((TIMER[9]>=0)) ;
1840:  !Fraeszeit ueberschritten ;
1841:  IF (F[329]),JMP LBL[2801] ;
1842:  !Umdrehungen Vergleichen ;
1843:  IF (R[1]<R[17]),JMP LBL[2800] ;
1844:  F[186]=(ON) ;
1845:  LBL[2801] ;
1846:  DO[1154]=((TIMER[9]<0)) ;
1847:  !Fraeser ausblasen EIN ;
1848:  DO[1167]=(F[330] OR (TIMER[9]<0)) ;
1849:  DO[1038]=(OFF) ;
1850:  !EZ3/SP3 oeffnen ;
1851:  DO[1037]=(!DI[1037]) ;
1852:  DO[18181]=(F[329]) ;
1853:  WAIT (!F[329] OR DI[26] OR DI[27])    ;
1854:  DO[18181]=(OFF) ;
1855:  DO[18181]=(ON) ;
1856:  WAIT (DI[1037])    ;
1857:  DO[18181]=(OFF) ;
1858:  DO[1037]=(OFF) ;
1859:  !Umdrehungen ruecksetzen ;
1860:  R[1]=0    ;
1861:  R[42]=28    ;
1862:  IF (F[329] OR F[325]),JMP LBL[28] ;
1863:  JMP LBL[29] ;
1864:   ;
1865:  !************************** ;
1866:  !*      Schritt 29        * ;
1867:  !* STAT EZ3/SP3 SF Teil 2 * ;
1868:  !************************** ;
1869:   ;
1870:  LBL[29] ;
1871:  R[41]=29    ;
1872:  !RSK gestartet ;
1873:  F[321]=(OFF) ;
1874:  F[329]=(OFF) ;
1875:  F[325]=(OFF) ;
1876:  DO[1038]=(OFF) ;
1877:  DO[1037]=(!DI[1037]) ;
1878:  DO[18181]=(ON) ;
1879:  WAIT (DI[1037])    ;
1880:  DO[18181]=(OFF) ;
1881:  DO[1154]=(ON) ;
1882:  DO[1037]=(OFF) ;
1883:  !EZ3/SP3 schliessen ;
1884:  DO[1038]=(ON) ;
1885:  !Fraeser ausblasen AUS/EIN ;
1886:  DO[1167]=(F[330]) ;
1887:  TIMER[9]=((-4)) ;
1888:  !EZ3/SP3 Kraft erreicht ;
1889:  WAIT ((DI[1038] AND !DI[1092] AND !DI[1100] AND !DI[1094] AND !DI[1095]) OR (TIMER[9]>=0))    ;
1890:  F[325]=((TIMER[9]>=0)) ;
1891:  DO[18181]=(ON) ;
1892:  DO[1038]=((TIMER[9]<0)) ;
1893:  DO[1154]=((TIMER[9]<0)) ;
1894:  WAIT ((DI[1038] AND !DI[1092] AND !DI[1100] AND !DI[1094] AND !DI[1095]) OR DI[26] OR DI[27])    ;
1895:  DO[18181]=(OFF) ;
1896:  !EZ3/SP3 Fehler Kraftaufbau ;
1897:  IF (F[325]),JMP LBL[2901] ;
1898:  TIMER[9]=((-5)) ;
1899:  LBL[2900] ;
1900:  WAIT (!DI[1154] OR F[325] OR (TIMER[9]>=0))    ;
1901:  WAIT (DI[1154] OR F[325] OR (TIMER[9]>=0))    ;
1902:  R[1]=(R[1]+1) ;
1903:  F[329]=((TIMER[9]>=0)) ;
1904:  !Fraeszeit ueberschritten ;
1905:  IF (F[329]),JMP LBL[2901] ;
1906:  !Umdrehungen Vergleichen ;
1907:  IF (R[1]<R[18]),JMP LBL[2900] ;
1908:  F[188]=(ON) ;
1909:  LBL[2901] ;
1910:  DO[1154]=((TIMER[9]<0)) ;
1911:  !Fraeser ausblasen EIN ;
1912:  DO[1167]=PULSE,4.0sec ;
1913:  DO[1038]=(OFF) ;
1914:  !EZ3/SP3 oeffnen ;
1915:  DO[1037]=(!DI[1037]) ;
1916:  DO[18181]=(F[329]) ;
1917:  WAIT (!F[329] OR DI[26] OR DI[27])    ;
1918:  DO[18181]=(OFF) ;
1919:  DO[18181]=(ON) ;
1920:  WAIT (DI[1037])    ;
1921:  DO[18181]=(OFF) ;
1922:  DO[1037]=(OFF) ;
1923:  !Umdrehungen ruecksetzen ;
1924:  R[1]=0    ;
1925:  R[42]=29    ;
1926:  IF (F[329] OR F[325]),JMP LBL[29] ;
1927:  JMP LBL[31] ;
1928:   ;
1929:  !******************* ;
1930:  !*   Schritt 30    * ;
1931:  !* STAT EZ3/SP3 NF * ;
1932:  !******************* ;
1933:   ;
1934:  LBL[30] ;
1935:  R[41]=30    ;
1936:  !RSK gestartet ;
1937:  F[321]=(OFF) ;
1938:  F[329]=(OFF) ;
1939:  F[325]=(OFF) ;
1940:  !Zähler wegspeichern für 2ten Hub ;
1941:  R[45]=R[19]    ;
1942:  IF (F[190] AND F[732]),R[19]=R[38] ;
1943:  DO[1038]=(OFF) ;
1944:  DO[1037]=(!DI[1037]) ;
1945:  DO[18181]=(ON) ;
1946:  WAIT (DI[1037])    ;
1947:  DO[18181]=(OFF) ;
1948:  DO[1154]=(ON) ;
1949:  DO[1037]=(OFF) ;
1950:  !EZ3/SP3 schliessen ;
1951:  DO[1038]=(ON) ;
1952:  !Fraeser ausblasen AUS ;
1953:  DO[1167]=(F[330]) ;
1954:  TIMER[9]=((-4)) ;
1955:  !EZ3/SP3 Kraft erreicht ;
1956:  WAIT ((DI[1038] AND !DI[1092] AND !DI[1100] AND !DI[1094] AND !DI[1095]) OR (TIMER[9]>=0))    ;
1957:  F[325]=((TIMER[9]>=0)) ;
1958:  DO[18181]=(ON) ;
1959:  DO[1038]=((TIMER[9]<0)) ;
1960:  DO[1154]=((TIMER[9]<0)) ;
1961:  WAIT ((DI[1038] AND !DI[1092] AND !DI[1100] AND !DI[1094] AND !DI[1095]) OR DI[26] OR DI[27])    ;
1962:  DO[18181]=(OFF) ;
1963:  !EZ3/SP3 Fehler Kraftaufbau ;
1964:  IF (F[325]),JMP LBL[3001] ;
1965:  TIMER[9]=((-5)) ;
1966:  LBL[3000] ;
1967:  WAIT (!DI[1154] OR F[325] OR (TIMER[9]>=0))    ;
1968:  WAIT (DI[1154] OR F[325] OR (TIMER[9]>=0))    ;
1969:  R[1]=(R[1]+1) ;
1970:  F[329]=((TIMER[9]>=0)) ;
1971:  !Fraeszeit ueberschritten ;
1972:  IF (F[329]),JMP LBL[3001] ;
1973:  !Umdrehungen Vergleichen ;
1974:  IF (R[1]<R[19]),JMP LBL[3000] ;
1975:  !EZ3/SP3 2 Huebe bei NF ;
1976:  IF (!F[200]),JMP LBL[3001] ;
1977:  IF (F[190]),F[188]=(ON) ;
1978:  F[190]=(ON) ;
1979:  LBL[3001] ;
1980:  DO[1154]=((TIMER[9]<0)) ;
1981:  !Fraeser ausblasen EIN ;
1982:  DO[1167]=PULSE,4.0sec ;
1983:  !EZ3/SP3 oeffnen ;
1984:  DO[1038]=(OFF) ;
1985:  DO[1037]=(!DI[1037]) ;
1986:  DO[18181]=(F[329]) ;
1987:  WAIT (!F[329] OR DI[26] OR DI[27])    ;
1988:  DO[18181]=(OFF) ;
1989:  DO[18181]=(ON) ;
1990:  WAIT (DI[1037])    ;
1991:  DO[18181]=(OFF) ;
1992:  DO[1037]=(OFF) ;
1993:  !Umdrehungen ruecksetzen ;
1994:  R[1]=0    ;
1995:  R[42]=30    ;
1996:  IF (F[190] AND F[732]),GO[3]=36 ;
1997:  IF (F[188] AND F[732]),R[19]=R[45] ;
1998:  IF (F[329] OR F[325] OR (!F[188] AND F[200])),JMP LBL[30] ;
1999:  F[190]=(ON) ;
2000:  JMP LBL[31] ;
2001:   ;
2002:  !**************************** ;
2003:  !*        Schritt 31        * ;
2004:  !* STAT EZ3/SP3 i.O./n.i.O. * ;
2005:  !**************************** ;
2006:   ;
2007:  LBL[31] ;
2008:  R[41]=31    ;
2009:  !Fraesueberwachung starten ;
2010:  TIMER[7]=((-5)) ;
2011:  WAIT ((F[174] OR F[175]) AND (F[190] OR (F[186] AND F[188])) OR (TIMER[7]>=0))    ;
2012:  F[329]=((TIMER[7]>=0)) ;
2013:  IF (!F[329]),R[41]=32 ;
2014:  IF (F[329]),R[41]=30 ;
2015:  !KF1 U-Merker ruecksetzen ;
2016:  F[186]=(OFF) ;
2017:  F[188]=(OFF) ;
2018:  F[190]=(OFF) ;
2019:  R[42]=31    ;
2020:  JMP LBL[R[41]] ;
2021:   ;
2022:  !**************************** ;
2023:  !*       Schritt 32         * ;
2024:  !*      STAT EZ3/SP3        * ;
2025:  !* KS3 in Ruhest. schwenken * ;
2026:  !**************************** ;
2027:   ;
2028:  LBL[32] ;
2029:  R[41]=32    ;
2030:  !RSK gestartet ;
2031:  F[321]=(OFF) ;
2032:  DO[1038]=(OFF) ;
2033:  DO[1037]=(!DI[1037]) ;
2034:  DO[18181]=(ON) ;
2035:  WAIT (DI[1037])    ;
2036:  DO[18181]=(OFF) ;
2037:  DO[1037]=(OFF) ;
2038:  TIMER[8]=((-4)) ;
2039:  WAIT ((DI[1164] AND !DI[1162] AND !DI[1165] AND DI[1163]) OR (TIMER[8]>=0))    ;
2040:  F[324]=((TIMER[8]>=0)) ;
2041:  DO[18181]=((TIMER[8]>=0)) ;
2042:  WAIT (DI[1164] AND !DI[1162] AND !DI[1165] AND DI[1163])    ;
2043:  DO[18181]=(OFF) ;
2044:  F[324]=(OFF) ;
2045:  TIMER[8]=((-4)) ;
2046:  DO[1155]=(F[564]) ;
2047:  WAIT ((DI[1155] AND F[564]) OR (!DI[1155] AND !F[564]) OR (TIMER[8]>=0))    ;
2048:  F[323]=((TIMER[8]>=0)) ;
2049:  DO[18181]=((TIMER[8]>=0)) ;
2050:  WAIT ((DI[1155] AND F[564]) OR (!DI[1155] AND !F[564]))    ;
2051:  DO[18181]=(OFF) ;
2052:  F[323]=(OFF) ;
2053:  !Ueberwachungszeit KS3 Schwenken ;
2054:  TIMER[8]=((-4)) ;
2055:  DO[3971]=(ON) ;
2056:  WAIT (DI[1161] OR (TIMER[8]>=0))    ;
2057:  DO[18181]=((TIMER[8]>=0)) ;
2058:  WAIT (DI[1161])    ;
2059:  TIMER[8]=((-6)) ;
2060:  DO[18181]=(OFF) ;
2061:  WAIT ((!DI[1164] AND DI[1162] AND DI[1165] AND !DI[1163]) OR (TIMER[8]>=0))    ;
2062:  F[323]=((TIMER[8]>=0)) ;
2063:  DO[3971]=(OFF) ;
2064:  DO[18181]=((TIMER[8]>=0)) ;
2065:  WAIT ((!DI[1164] AND DI[1162] AND DI[1165] AND !DI[1163]) OR DI[26])    ;
2066:  DO[18181]=(OFF) ;
2067:  F[323]=(OFF) ;
2068:  DO[1154]=(OFF) ;
2069:  DO[1155]=(OFF) ;
2070:  !Sprung zurueck bei KS3 Fehler ;
2071:  IF (TIMER[8]>=0),JMP LBL[32] ;
2072:  R[42]=32    ;
2073:  JMP LBL[33] ;
2074:   ;
2075:  !*********************** ;
2076:  !*     Schritt 33      * ;
2077:  !*    STAT EZ3/SP3     * ;
2078:  !* Messen nach Fraesen * ;
2079:  !*********************** ;
2080:   ;
2081:  LBL[33] ;
2082:  R[41]=33    ;
2083:  !RSK gestartet ;
2084:  F[321]=(OFF) ;
2085:  GO[9]=1 ;
2086:  WAIT    .10(sec) ;
2087:  DO[1106]=(ON) ;
2088:  !STAT EZ3/SP3 FK Fraesen ;
2089:  DO[18181]=(ON) ;
2090:  WAIT (!DI[1106] AND DI[1107] AND !DI[1108])    ;
2091:  DO[18181]=(OFF) ;
2092:  DO[1106]=(OFF) ;
2093:  GO[7]=(31) ;
2094:  GO[9]=(31) ;
2095:  WAIT    .10(sec) ;
2096:  DO[1077]=(ON) ;
2097:  TIMER[9]=((-8)) ;
2098:  WAIT (DI[1077] OR (TIMER[9]>=0))    ;
2099:  DO[326]=((TIMER[9]>=0)) ;
2100:  DO[18181]=(ON) ;
2101:  WAIT (DI[1077] OR DI[26] OR DI[27])    ;
2102:  DO[18181]=(OFF) ;
2103:  DO[326]=(OFF) ;
2104:  F[179]=(DI[1096] OR DI[1097]) ;
2105:  DO[1077]=(OFF) ;
2106:  F[180]=(DI[1056] OR (DI[1055] AND DI[1054] AND DI[1053])) ;
2107:  TIMER[7]=((-2)) ;
2108:  WAIT ((!F[180] AND !F[179]) OR (TIMER[7]>=0))    ;
2109:  F[329]=((TIMER[7]>=0)) ;
2110:  DO[18181]=(F[329]) ;
2111:  WAIT ((!F[180] AND !F[179]) OR DI[26] OR DI[27])    ;
2112:  DO[18181]=(OFF) ;
2113:  F[329]=(OFF) ;
2114:  F[298]=(F[180] OR F[179]) ;
2115:  DO[1037]=(!DI[1037]) ;
2116:  DO[18181]=(ON) ;
2117:  WAIT ((DI[1037] AND !DI[1104]) OR (DI[1037] AND F[298]))    ;
2118:  DO[18181]=(OFF) ;
2119:  DO[1037]=(OFF) ;
2120:  R[42]=33    ;
2121:  !EZ3/SP3 wiederh. bei Messfehler ;
2122:  IF (F[298]),JMP LBL[27] ;
2123:  DO[1078]=(OFF) ;
2124:  DO[1079]=(OFF) ;
2125:  !KS nicht bei K-Verschleiss ;
2126:  IF (DI[1097]),JMP LBL[35] ;
2127:  !EZ3/SP3 2.Setzhub nach Fraesen ;
2128:  IF (F[335] AND F[174]),JMP LBL[57] ;
2129:  !EZ3/SP3 Kurzschluss schweissen ;
2130:  IF (F[335] AND !F[174]),JMP LBL[34] ;
2131:  !EZ3/SP3 Kurzschluss schweissen ;
2132:  IF (!F[335]),JMP LBL[34] ;
2133:   ;
2134:  !************************** ;
2135:  !*      Schritt 34        * ;
2136:  !*     STAT EZ3/SP3       * ;
2137:  !* Kurzschlussschweissung * ;
2138:  !************************** ;
2139:   ;
2140:  LBL[34] ;
2141:  R[41]=34    ;
2142:  !RSK gestartet ;
2143:  F[321]=(OFF) ;
2144:  DO[209]=(ON) ;
2145:  !EZ3/SP3/SK3 Prog. ;
2146:  IF (F[174] AND !F[301]),GO[7]=(41) ;
2147:  IF (F[174] AND !F[301]),GO[9]=(41) ;
2148:  IF (F[175] OR F[301]),GO[7]=(51) ;
2149:  IF (F[175] OR F[301]),GO[9]=(51) ;
2150:  WAIT    .10(sec) ;
2151:  DO[1037]=(OFF) ;
2152:  DO[1038]=(OFF) ;
2153:  DO[1105]=(OFF) ;
2154:  DO[514]=(OFF) ;
2155:  F[176]=(OFF) ;
2156:  F[306]=(OFF) ;
2157:  F[303]=(!DI[1089] AND DI[1104]) ;
2158:  DO[18181]=(ON) ;
2159:  WAIT (DI[1025] AND DI[1033] AND DI[1034] AND (!DI[1104] OR (DI[1089] AND DI[1104])))    ;
2160:  DO[18181]=(OFF) ;
2161:  F[303]=(OFF) ;
2162:  DO[18181]=(ON) ;
2163:  WAIT ((!DI[1105] AND DI[1112] AND DI[1122] AND !F[176]) OR (!DI[1112] AND DI[1122] AND DI[209]))    ;
2164:  DO[18181]=(OFF) ;
2165:  !EZ3/SP3 schliessen ;
2166:  DO[1038]=(ON) ;
2167:  TIMER[9]=((-4)) ;
2168:  !EZ3/SP3 Kraft erreicht ;
2169:  WAIT ((DI[1038] AND !DI[1092] AND !DI[1100]) OR DI[1094] OR DI[1095] OR (TIMER[9]>=0))    ;
2170:  DO[1038]=(DI[1038] AND !DI[1094] AND !DI[1095]) ;
2171:  DO[1037]=(!DO[1038]) ;
2172:  !Schweissen START ;
2173:  DO[1105]=(DI[1038] AND !DI[1094] AND !DI[1095]) ;
2174:  !EZ3/SP3 Fehler Ausgleich ;
2175:  F[302]=(DI[1038] AND DI[1039]) ;
2176:  !EZ3/SP3 Fehler SZ ;
2177:  F[300]=(DI[1094] OR DI[1095]) ;
2178:  !SK3 FK ;
2179:  TIMER[9]=((-10)) ;
2180:  WAIT ((F[176] AND DO[1105]) OR ((DI[1124] OR DI[1125]) AND (DI[1105] AND DO[1105])) OR (DI[1091] AND DI[1104]) OR !DO[1105] OR (TIMER[9]>=0))    ;
2181:  F[297]=(F[176] OR (DI[1124] AND !DI[1126] AND !DI[1095] AND DI[1105])) ;
2182:  !SK3 Fehler ;
2183:  F[301]=(!F[297] AND !F[298] AND DO[1105]) ;
2184:  DO[1105]=(OFF) ;
2185:  DO[1038]=(OFF) ;
2186:  DO[18181]=(ON) ;
2187:  F[749]=(!F[297] AND !F[748]) ;
2188:  F[748]=(!F[297]) ;
2189:  WAIT (F[297] OR DI[26] OR DI[27] OR (F[749] AND F[731]))    ;
2190:  WAIT (!DI[26] AND !DI[27])    ;
2191:  DO[18181]=(OFF) ;
2192:  !EZ3/SP3 oeffnen ;
2193:  DO[1037]=(!DI[1037]) ;
2194:  DO[18181]=(ON) ;
2195:  WAIT (DI[1037])    ;
2196:  DO[18181]=(OFF) ;
2197:  DO[1037]=(OFF) ;
2198:  F[303]=(OFF) ;
2199:  DO[209]=(OFF) ;
2200:  R[42]=34    ;
2201:  JMP LBL[35] ;
2202:   ;
2203:  !************************** ;
2204:  !*       Schritt 35       * ;
2205:  !*      STAT EZ3/SP3      * ;
2206:  !************************** ;
2207:   ;
2208:  LBL[35] ;
2209:  R[41]=35    ;
2210:  !RSK gestartet ;
2211:  F[321]=(OFF) ;
2212:  !Sprung zurueck bei Fehler ;
2213:  IF (!F[297] AND !DI[1097]),JMP LBL[27] ;
2214:  !STAT EZ3/SP3 FK Fraesen ;
2215:  F[185]=(!F[329]) ;
2216:  DO[116]=(OFF) ;
2217:  DO[194]=(OFF) ;
2218:  R[42]=35    ;
2219:  JMP LBL[1] ;
2220:   ;
2221:   ;
2222:  !***************** ;
2223:  !***************** ;
2224:  !* MS1 Reinigung * ;
2225:  !***************** ;
2226:  !***************** ;
2227:   ;
2228:   ;
2229:  !******************************* ;
2230:  !*         Schritt 36          * ;
2231:  !*       MS1 Reinigung         * ;
2232:  !* KS3 in Arbeitsst. schwenken * ;
2233:  !******************************* ;
2234:   ;
2235:  LBL[36] ;
2236:  R[41]=36    ;
2237:  !RSK gestartet ;
2238:  F[321]=(OFF) ;
2239:  !MS bei Reinigung ;
2240:  DO[116]=(ON) ;
2241:  !Reinigung MS1 gestartet ;
2242:  F[604]=(ON) ;
2243:  !Ueberwachungszeit KS3 ;
2244:  TIMER[8]=((-4)) ;
2245:  WAIT ((!DI[1164] AND DI[1162] AND DI[1165] AND !DI[1163]) OR (TIMER[8]>=0))    ;
2246:  F[323]=((TIMER[8]>=0)) ;
2247:  DO[18181]=((TIMER[8]>=0)) ;
2248:  WAIT (!DI[1164] AND DI[1162] AND DI[1165] AND !DI[1163])    ;
2249:  DO[18181]=(OFF) ;
2250:  F[323]=(OFF) ;
2251:  !KS3 in Arbeitsst. schwenken ;
2252:  TIMER[8]=((-4)) ;
2253:  DO[3974]=(ON) ;
2254:  WAIT (DI[1161] OR (TIMER[8]>=0))    ;
2255:  DO[18181]=((TIMER[8]>=0)) ;
2256:  WAIT (DI[1161])    ;
2257:  DO[18181]=(OFF) ;
2258:  TIMER[8]=((-6)) ;
2259:  WAIT ((DI[1164] AND !DI[1162] AND !DI[1165] AND DI[1163]) OR (TIMER[8]>=0))    ;
2260:  F[324]=((TIMER[8]>=0)) ;
2261:  DO[3974]=(OFF) ;
2262:  DO[18181]=((TIMER[8]>=0)) ;
2263:  WAIT ((DI[1164] AND !DI[1162] AND !DI[1165] AND DI[1163]) OR DI[26])    ;
2264:  DO[18181]=(OFF) ;
2265:  F[324]=(OFF) ;
2266:  !Sprung bei Fehler KS3 schwenken ;
2267:  IF (TIMER[8]>=0),JMP LBL[36] ;
2268:  R[42]=36    ;
2269:  JMP LBL[37] ;
2270:   ;
2271:  !*************************** ;
2272:  !*      Schritt 37         * ;
2273:  !* MS1 Reinigung starten   * ;
2274:  !*************************** ;
2275:   ;
2276:  LBL[37] ;
2277:  R[41]=37    ;
2278:  TIMER[9]=((-2)) ;
2279:  WAIT ((DI[10] AND DI[13] AND DI[23]) OR (TIMER[9]>=0))    ;
2280:  F[329]=((TIMER[9]>=0)) ;
2281:  DO[18181]=((TIMER[9]>=0)) ;
2282:  WAIT (DI[10] AND DI[13] AND DI[23])    ;
2283:  F[329]=(OFF) ;
2284:  DO[18181]=(OFF) ;
2285:  !MS1 Reinigung i.O. ;
2286:  DO[18181]=(ON) ;
2287:  WAIT (DI[1864])    ;
2288:  DO[18181]=(OFF) ;
2289:  !MS1 Ausblasen EIN ;
2290:  DO[1870]=(ON) ;
2291:  !MS1 Reinigung EIN ;
2292:  TIMER[9]=((-1)) ;
2293:  DO[1864]=(ON) ;
2294:  !Einschaltdauer Reingung ;
2295:  TIMER[7]=((R[26])) ;
2296:  WAIT (!DI[1864] OR (TIMER[9]>=0))    ;
2297:  F[329]=((TIMER[9]>=0)) ;
2298:  DO[18181]=((TIMER[9]>=0)) ;
2299:  WAIT (!DI[1864] OR DI[26])    ;
2300:  WAIT ((TIMER[7]>=0))    ;
2301:  F[329]=(OFF) ;
2302:  DO[18181]=(OFF) ;
2303:  !MS1 Reinigung AUS ;
2304:  DO[1864]=(OFF) ;
2305:  TIMER[9]=((-6)) ;
2306:  WAIT (DI[1864] OR (TIMER[9]>=0))    ;
2307:  F[329]=((TIMER[9]>=0)) ;
2308:  DO[18181]=((TIMER[9]>=0)) ;
2309:  WAIT (DI[1864] OR DI[26] OR !DI[13] OR !DI[23])    ;
2310:  IF (DI[26] OR !DI[13] OR !DI[23]),JMP LBL[37] ;
2311:  F[329]=(OFF) ;
2312:  DO[18181]=(OFF) ;
2313:  !MS1 Ausblasen AUS ;
2314:  DO[1870]=(OFF) ;
2315:  !MS1 Einspruehen ;
2316:  TIMER[9]=((R[23])) ;
2317:  DO[520]=(!F[574] AND F[575]) ;
2318:  DO[1871]=(F[574] AND F[575]) ;
2319:  WAIT (!F[575] OR (TIMER[9]>=0))    ;
2320:  DO[520]=(OFF) ;
2321:  DO[1871]=(OFF) ;
2322:  R[42]=37    ;
2323:  JMP LBL[38] ;
2324:   ;
2325:  !**************************** ;
2326:  !*          Schritt 38      * ;
2327:  !*       MS1 Reinigung      * ;
2328:  !* KS3 in Ruhest. schwenken * ;
2329:  !**************************** ;
2330:   ;
2331:  LBL[38] ;
2332:  R[41]=38    ;
2333:  !Ueberwachungszeit KS3 ;
2334:  TIMER[8]=((-4)) ;
2335:  WAIT ((DI[1164] AND !DI[1162] AND !DI[1165] AND DI[1163]) OR (TIMER[8]>=0))    ;
2336:  F[324]=((TIMER[8]>=0)) ;
2337:  DO[18181]=((TIMER[8]>=0)) ;
2338:  WAIT (DI[1164] AND !DI[1162] AND !DI[1165] AND DI[1163])    ;
2339:  DO[18181]=(OFF) ;
2340:  F[324]=(OFF) ;
2341:  !KS3 in Ruhestest. schwenken ;
2342:  TIMER[8]=((-4)) ;
2343:  DO[3971]=(ON) ;
2344:  WAIT (DI[1161] OR (TIMER[8]>=0))    ;
2345:  DO[18181]=((TIMER[8]>=0)) ;
2346:  WAIT (DI[1161])    ;
2347:  DO[18181]=(OFF) ;
2348:  TIMER[8]=((-6)) ;
2349:  WAIT ((!DI[1164] AND DI[1162] AND DI[1165] AND !DI[1163]) OR (TIMER[8]>=0))    ;
2350:  F[323]=((TIMER[8]>=0)) ;
2351:  DO[3971]=(OFF) ;
2352:  DO[18181]=((TIMER[8]>=0)) ;
2353:  WAIT ((!DI[1164] AND DI[1162] AND DI[1165] AND !DI[1163]) OR DI[26])    ;
2354:  DO[18181]=(OFF) ;
2355:  F[323]=(OFF) ;
2356:  !Sprung bei Fehler KS3 schwenken ;
2357:  IF (TIMER[8]>=0),JMP LBL[38] ;
2358:  R[42]=38    ;
2359:  JMP LBL[39] ;
2360:   ;
2361:  !***************************** ;
2362:  !*         Schritt 39        * ;
2363:  !* MS1 Reinigung ruecksetzen * ;
2364:  !***************************** ;
2365:   ;
2366:  LBL[39] ;
2367:  R[41]=39    ;
2368:  !MS1 Zaehler ruecksetzen ;
2369:  R[21]=0    ;
2370:  !MS FRG Reinigung ;
2371:  F[603]=(OFF) ;
2372:  !MS1 Reinigung FK ;
2373:  F[605]=(ON) ;
2374:  R[42]=39    ;
2375:  JMP LBL[1] ;
2376:   ;
2377:   ;
2378:  !***************** ;
2379:  !***************** ;
2380:  !* MS2 Reinigung * ;
2381:  !***************** ;
2382:  !***************** ;
2383:   ;
2384:   ;
2385:  !******************************* ;
2386:  !*         Schritt 40          * ;
2387:  !*       MS2 Reinigung         * ;
2388:  !* KS2 in Arbeitsst. schwenken * ;
2389:  !******************************* ;
2390:   ;
2391:  LBL[40] ;
2392:  R[41]=40    ;
2393:  !RSK gestartet ;
2394:  F[321]=(OFF) ;
2395:  !Reinigung MS2 gestartet ;
2396:  F[608]=(ON) ;
2397:  !MS bei Reinigung ;
2398:  DO[116]=(ON) ;
2399:  !Ueberwachungszeit KS2 ;
2400:  TIMER[8]=((-4)) ;
2401:  WAIT ((!DI[1004] AND DI[1002] AND DI[1005] AND !DI[1003]) OR (TIMER[8]>=0))    ;
2402:  F[323]=((TIMER[8]>=0)) ;
2403:  DO[18181]=((TIMER[8]>=0)) ;
2404:  WAIT (!DI[1004] AND DI[1002] AND DI[1005] AND !DI[1003])    ;
2405:  DO[18181]=(OFF) ;
2406:  F[323]=(OFF) ;
2407:  !KS2 in Arbeitsst. schwenken ;
2408:  TIMER[8]=((-4)) ;
2409:  DO[3973]=(ON) ;
2410:  WAIT (DI[1001] OR (TIMER[8]>=0))    ;
2411:  DO[18181]=((TIMER[8]>=0)) ;
2412:  WAIT (DI[1001])    ;
2413:  DO[18181]=(OFF) ;
2414:  TIMER[8]=((-4)) ;
2415:  WAIT ((DI[1004] AND !DI[1002] AND !DI[1005] AND DI[1003]) OR (TIMER[8]>=0))    ;
2416:  F[324]=((TIMER[8]>=0)) ;
2417:  DO[3973]=(OFF) ;
2418:  DO[18181]=((TIMER[8]>=0)) ;
2419:  WAIT ((DI[1004] AND !DI[1002] AND !DI[1005] AND DI[1003]) OR DI[26])    ;
2420:  DO[18181]=(OFF) ;
2421:  F[324]=(OFF) ;
2422:  !Sprung bei Fehler KS2 schwenken ;
2423:  IF (TIMER[8]>=0),JMP LBL[40] ;
2424:  R[42]=40    ;
2425:  JMP LBL[41] ;
2426:   ;
2427:  !*************************** ;
2428:  !*      Schritt 41         * ;
2429:  !* MS2 Reinigung starten   * ;
2430:  !*************************** ;
2431:   ;
2432:  LBL[41] ;
2433:  R[41]=41    ;
2434:  TIMER[9]=((-2)) ;
2435:  WAIT ((DI[10] AND DI[13] AND DI[23]) OR (TIMER[9]>=0))    ;
2436:  F[329]=((TIMER[9]>=0)) ;
2437:  DO[18181]=((TIMER[9]>=0)) ;
2438:  WAIT (DI[10] AND DI[13] AND DI[23])    ;
2439:  F[329]=(OFF) ;
2440:  DO[18181]=(OFF) ;
2441:  !MS2 Ausblasen EIN ;
2442:  DO[1902]=(ON) ;
2443:  !MS2 Reinigung EIN ;
2444:  TIMER[9]=((-1)) ;
2445:  DO[1896]=(ON) ;
2446:  WAIT (!DI[1896] OR (TIMER[9]>=0))    ;
2447:  F[329]=((TIMER[9]>=0)) ;
2448:  DO[18181]=((TIMER[9]>=0)) ;
2449:  WAIT (!DI[1896] OR DI[26])    ;
2450:  F[329]=(OFF) ;
2451:  DO[18181]=(OFF) ;
2452:  !MS2 Reinigung AUS ;
2453:  DO[1896]=(OFF) ;
2454:  TIMER[9]=((-6)) ;
2455:  WAIT (DI[1896] OR (TIMER[9]>=0))    ;
2456:  F[329]=((TIMER[9]>=0)) ;
2457:  DO[18181]=((TIMER[9]>=0)) ;
2458:  WAIT (DI[1896] OR DI[26] OR !DI[13] OR !DI[23])    ;
2459:  IF (DI[26] OR !DI[13] OR !DI[23]),JMP LBL[41] ;
2460:  F[329]=(OFF) ;
2461:  DO[18181]=(OFF) ;
2462:  !MS2 Ausblasen AUS ;
2463:  DO[1902]=(OFF) ;
2464:  !MS2 Einspruehen ;
2465:  TIMER[9]=((R[23])) ;
2466:  DO[528]=(!F[583] AND F[584]) ;
2467:  DO[1903]=(F[583] AND F[585]) ;
2468:  WAIT (!F[584] OR (TIMER[9]>=0))    ;
2469:  DO[528]=(OFF) ;
2470:  DO[1903]=(OFF) ;
2471:  R[42]=41    ;
2472:  JMP LBL[42] ;
2473:   ;
2474:  !**************************** ;
2475:  !*          Schritt 42      * ;
2476:  !*       MS2 Reinigung      * ;
2477:  !* KS2 in Ruhest. schwenken * ;
2478:  !**************************** ;
2479:   ;
2480:  LBL[42] ;
2481:  R[41]=42    ;
2482:  !Ueberwachungszeit KS2 ;
2483:  TIMER[8]=((-4)) ;
2484:  WAIT ((DI[1004] AND !DI[1002] AND !DI[1005] AND DI[1003]) OR (TIMER[8]>=0))    ;
2485:  F[324]=((TIMER[8]>=0)) ;
2486:  DO[18181]=((TIMER[8]>=0)) ;
2487:  WAIT (DI[1004] AND !DI[1002] AND !DI[1005] AND DI[1003])    ;
2488:  DO[18181]=(OFF) ;
2489:  F[324]=(OFF) ;
2490:  !KS2 in Ruhestest. schwenken ;
2491:  TIMER[8]=((-4)) ;
2492:  DO[3970]=(ON) ;
2493:  WAIT (DI[1001] OR (TIMER[8]>=0))    ;
2494:  DO[18181]=((TIMER[8]>=0)) ;
2495:  WAIT (DI[1001])    ;
2496:  DO[18181]=(OFF) ;
2497:  TIMER[8]=((-6)) ;
2498:  WAIT ((!DI[1004] AND DI[1002] AND DI[1005] AND !DI[1003]) OR (TIMER[8]>=0))    ;
2499:  F[323]=((TIMER[8]>=0)) ;
2500:  DO[3970]=(OFF) ;
2501:  DO[18181]=((TIMER[8]>=0)) ;
2502:  WAIT ((!DI[1004] AND DI[1002] AND DI[1005] AND !DI[1003]) OR DI[26])    ;
2503:  DO[18181]=(OFF) ;
2504:  F[323]=(OFF) ;
2505:  !Sprung bei Fehler KS2 schwenken ;
2506:  IF (TIMER[8]>=0),JMP LBL[42] ;
2507:  R[42]=42    ;
2508:  JMP LBL[43] ;
2509:   ;
2510:  !***************************** ;
2511:  !*         Schritt 43        * ;
2512:  !* MS2 Reinigung ruecksetzen * ;
2513:  !***************************** ;
2514:   ;
2515:  LBL[43] ;
2516:  R[41]=43    ;
2517:  !MS2 Zaehler ruecksetzen ;
2518:  R[22]=0    ;
2519:  !MS2 FRG Reinigung ;
2520:  F[607]=(OFF) ;
2521:  !MS2 Reinigung FK ;
2522:  F[609]=(ON) ;
2523:  R[42]=43    ;
2524:  JMP LBL[1] ;
2525:   ;
2526:  !******************************** ;
2527:  !*            Schritt 44 ;
2528:  !*          KL1 Spueleimer ;
2529:  !*  (an Pneum. Schwenkeinheit KL1 ;
2530:  !*     KL1 in Arbeitsst. schwenke ;
2531:  !******************************** ;
2532:   ;
2533:  LBL[44] ;
2534:  R[41]=44    ;
2535:  !RSK gestartet ;
2536:  F[321]=(OFF) ;
2537:  DO[161]=(ON) ;
2538:  !Steuerluft EIN ;
2539:  DO[2113]=(ON) ;
2540:  TIMER[9]=((-2)) ;
2541:  !Warte auf Vorwahl Ventilinsel ;
2542:  WAIT ((F[523] AND !F[524]) OR (!F[523] AND F[524]) OR (TIMER[9]>=0))    ;
2543:  DO[120]=(TIMER[9]>=0) ;
2544:  DO[18181]=((TIMER[9]>=0)) ;
2545:  WAIT ((F[523] AND !F[524]) OR (!F[523] AND F[524]))    ;
2546:  DO[120]=(OFF) ;
2547:  DO[18181]=(OFF) ;
2548:  !WAIT Steuerluft EIN ;
2549:  WAIT ((F[523] AND !F[524] AND DI[2113]) OR (!F[523] AND F[524] AND !DI[2114]) OR (TIMER[9]>=0))    ;
2550:  DO[120]=(TIMER[9]>=0) ;
2551:  DO[18181]=((TIMER[9]>=0)) ;
2552:  WAIT ((F[523] AND !F[524] AND DI[2113]) OR (!F[523] AND F[524] AND !DI[2114]))    ;
2553:  DO[120]=(OFF) ;
2554:  DO[18181]=(OFF) ;
2555:  !In Arbeitsstellung schwenken ;
2556:  DO[2115]=(OFF) ;
2557:  DO[2116]=(ON) ;
2558:  !Freigabe Bewegung (ON) ;
2559:  DO[2117]=(OFF) ;
2560:  DO[2118]=(ON) ;
2561:  TIMER[9]=((-10)) ;
2562:  !Warte bis Spueleimer in Position ;
2563:  WAIT ((!DI[2115] AND DI[2116]) OR (TIMER[9]>=0))    ;
2564:  DO[120]=(TIMER[9]>=0) ;
2565:  DO[18181]=((TIMER[9]>=0)) ;
2566:  WAIT (!DI[2115] AND DI[2116])    ;
2567:  DO[120]=(OFF) ;
2568:  DO[18181]=(OFF) ;
2569:  F[355]=((!DI[2115] AND DI[2116]) OR (F[837])) ;
2570:  WAIT    .30(sec) ;
2571:  !In Ruhestellung schwenken AUS ;
2572:  DO[2115]=(OFF) ;
2573:  !In Arbeitsstellung schw. AUS ;
2574:  DO[2116]=(OFF) ;
2575:  !Freigabe Bewegung AUS ;
2576:  DO[2118]=(OFF) ;
2577:  TIMER[9]=((-5)) ;
2578:  WAIT ((DI[2118]) OR (DI[2117] AND F[837]) OR (TIMER[9]>=0))    ;
2579:  DO[120]=(TIMER[9]>=0) ;
2580:  DO[18181]=((TIMER[9]>=0)) ;
2581:  WAIT ((DI[2118]) OR (DI[2117] AND F[837]))    ;
2582:  DO[120]=(OFF) ;
2583:  DO[18181]=(OFF) ;
2584:  !Freigabe  in  Endlage  halten ;
2585:  DO[2117]=(!F[837]) ;
2586:  IF (F[837]),DO[2118]=PULSE,0.5sec ;
2587:  TIMER[9]=((-10)) ;
2588:  WAIT ((DI[2117]) OR (DI[2118] AND F[837]) OR (TIMER[9]>=0))    ;
2589:  DO[120]=(TIMER[9]>=0) ;
2590:  DO[18181]=((TIMER[9]>=0)) ;
2591:  WAIT ((DI[2117]) OR (DI[2118] AND F[837]))    ;
2592:  DO[120]=(OFF) ;
2593:  DO[18181]=(OFF) ;
2594:  DO[161]=(OFF) ;
2595:  R[42]=44    ;
2596:  JMP LBL[1] ;
2597:   ;
2598:  !******************************** ;
2599:  !*           Schritt 45 ;
2600:  !*         KL1 Spueleimer ;
2601:  !* (an Pneum. Schwenkeinheit KL1) ;
2602:  !*    KL1 in Ruhest. schwenken ;
2603:  !******************************** ;
2604:   ;
2605:  LBL[45] ;
2606:  R[41]=45    ;
2607:  !RSK gestartet ;
2608:  F[321]=(OFF) ;
2609:  DO[161]=(ON) ;
2610:  !Steuerluft EIN ;
2611:  DO[2113]=(ON) ;
2612:  TIMER[9]=((-2)) ;
2613:  !Warte auf Vorwahl Ventilinsel ;
2614:  WAIT ((F[523] AND !F[524]) OR (!F[523] AND F[524]) OR (TIMER[9]>=0))    ;
2615:  DO[120]=(TIMER[9]>=0) ;
2616:  DO[18181]=((TIMER[9]>=0)) ;
2617:  WAIT ((F[523] AND !F[524]) OR (!F[523] AND F[524]))    ;
2618:  DO[120]=(OFF) ;
2619:  DO[18181]=(OFF) ;
2620:  !Warte bis Steuerluft EIN ;
2621:  WAIT ((F[523] AND !F[524] AND DI[2113]) OR (!F[523] AND F[524] AND !DI[2114]) OR (TIMER[9]>=0))    ;
2622:  DO[120]=(TIMER[9]>=0) ;
2623:  DO[18181]=((TIMER[9]>=0)) ;
2624:  WAIT ((F[523] AND !F[524] AND DI[2113]) OR (!F[523] AND F[524] AND !DI[2114]))    ;
2625:  DO[120]=(OFF) ;
2626:  DO[18181]=(OFF) ;
2627:  !In Ruhestellung schwenken EIN ;
2628:  DO[2115]=(ON) ;
2629:  DO[2116]=(OFF) ;
2630:  !Freigabe Bewegung EIN ;
2631:  DO[2117]=(OFF) ;
2632:  DO[2118]=(ON) ;
2633:  TIMER[9]=((-10)) ;
2634:  !Warte bis Spueleimer in Position ;
2635:  WAIT ((DI[2115] AND !DI[2116]) OR (TIMER[9]>=0))    ;
2636:  DO[120]=(TIMER[9]>=0) ;
2637:  DO[18181]=((TIMER[9]>=0)) ;
2638:  WAIT (DI[2115] AND !DI[2116])    ;
2639:  DO[120]=(OFF) ;
2640:  DO[18181]=(OFF) ;
2641:  F[355]=((DI[2115] AND !DI[2116]) OR (F[837])) ;
2642:  WAIT    .30(sec) ;
2643:  !In Ruhestellung schwenken AUS ;
2644:  DO[2115]=(OFF) ;
2645:  !In Arbeitsstellung schw. AUS ;
2646:  DO[2116]=(OFF) ;
2647:  !Freigabe Bewegung AUS ;
2648:  DO[2118]=(OFF) ;
2649:  TIMER[9]=((-5)) ;
2650:  WAIT ((DI[2118]) OR (DI[2117] AND F[837]) OR (TIMER[9]>=0))    ;
2651:  DO[120]=(TIMER[9]>=0) ;
2652:  DO[18181]=((TIMER[9]>=0)) ;
2653:  WAIT ((DI[2118]) OR (DI[2117] AND F[837]))    ;
2654:  DO[120]=(OFF) ;
2655:  DO[18181]=(OFF) ;
2656:  !Freigabe  in  Endlage  halten ;
2657:  DO[2117]=(!F[837]) ;
2658:  IF (F[837]),DO[2118]=PULSE,0.5sec ;
2659:  TIMER[9]=((-10)) ;
2660:  WAIT ((DI[2117]) OR (DI[2118] AND F[837]) OR (TIMER[9]>=0))    ;
2661:  DO[120]=(TIMER[9]>=0) ;
2662:  DO[18181]=((TIMER[9]>=0)) ;
2663:  WAIT ((DI[2117]) OR (DI[2118] AND F[837]))    ;
2664:  DO[120]=(OFF) ;
2665:  DO[18181]=(OFF) ;
2666:  DO[161]=(OFF) ;
2667:  R[42]=45    ;
2668:  JMP LBL[1] ;
2669:   ;
2670:  !******************************** ;
2671:  !*            Schritt 46 ;
2672:  !*          KL2 Spueleimer ;
2673:  !*  (an Pneum. Schwenkeinheit KL2 ;
2674:  !*     KL2 in Arbeitsst. schwenke ;
2675:  !******************************** ;
2676:   ;
2677:  LBL[46] ;
2678:  R[41]=46    ;
2679:  !RSK gestartet ;
2680:  F[321]=(OFF) ;
2681:  DO[177]=(ON) ;
2682:  !Steuerluft EIN ;
2683:  DO[2121]=(ON) ;
2684:  TIMER[9]=((-2)) ;
2685:  !Warte auf Vorwahl Ventilinsel ;
2686:  WAIT ((F[523] AND !F[524]) OR (!F[523] AND F[524]) OR (TIMER[9]>=0))    ;
2687:  DO[120]=(TIMER[9]>=0) ;
2688:  DO[18181]=((TIMER[9]>=0)) ;
2689:  WAIT ((F[523] AND !F[524]) OR (!F[523] AND F[524]))    ;
2690:  DO[120]=(OFF) ;
2691:  DO[18181]=(OFF) ;
2692:  !Warte Steuerluft EIN ;
2693:  WAIT ((F[523] AND !F[524] AND DI[2121]) OR (!F[523] AND F[524] AND !DI[2122]) OR (TIMER[9]>=0))    ;
2694:  DO[120]=(TIMER[9]>=0) ;
2695:  DO[18181]=((TIMER[9]>=0)) ;
2696:  WAIT ((F[523] AND !F[524] AND DI[2121]) OR (!F[523] AND F[524] AND !DI[2122]))    ;
2697:  DO[120]=(OFF) ;
2698:  DO[18181]=(OFF) ;
2699:  !In Arbeitsstellung schwenken EI ;
2700:  DO[2123]=(OFF) ;
2701:  DO[2124]=(ON) ;
2702:  !Freigabe Bewegung EIN ;
2703:  DO[2125]=(OFF) ;
2704:  DO[2126]=(ON) ;
2705:  TIMER[9]=((-10)) ;
2706:  !Warte bis Spueleimer in Position ;
2707:  WAIT ((!DI[2123] AND DI[2124]) OR (TIMER[9]>=0))    ;
2708:  DO[120]=(TIMER[9]>=0) ;
2709:  DO[18181]=((TIMER[9]>=0)) ;
2710:  WAIT (!DI[2123] AND DI[2124])    ;
2711:  DO[120]=(OFF) ;
2712:  DO[18181]=(OFF) ;
2713:  F[376]=(!DI[2123] AND DI[2124]) ;
2714:  WAIT    .30(sec) ;
2715:  !In Ruhestellung schwenken AUS ;
2716:  DO[2123]=(OFF) ;
2717:  !In Arbeitsstellung schwenken AU ;
2718:  DO[2124]=(OFF) ;
2719:  !Freigabe Bewegung AUS ;
2720:  DO[2126]=(OFF) ;
2721:  TIMER[9]=((-5)) ;
2722:  WAIT (DI[2126] OR (TIMER[9]>=0))    ;
2723:  DO[120]=(TIMER[9]>=0) ;
2724:  DO[18181]=((TIMER[9]>=0)) ;
2725:  WAIT (DI[2126])    ;
2726:  DO[120]=(OFF) ;
2727:  DO[18181]=(OFF) ;
2728:  !Freigabe  in  Endlage  halten ;
2729:  DO[2125]=(ON) ;
2730:  TIMER[9]=((-10)) ;
2731:  WAIT (DI[2125] OR (TIMER[9]>=0))    ;
2732:  DO[120]=(TIMER[9]>=0) ;
2733:  DO[18181]=((TIMER[9]>=0)) ;
2734:  WAIT (DI[2125])    ;
2735:  DO[120]=(OFF) ;
2736:  DO[18181]=(OFF) ;
2737:  DO[177]=(OFF) ;
2738:  R[42]=46    ;
2739:  JMP LBL[1] ;
2740:   ;
2741:  !******************************** ;
2742:  !*           Schritt 47 ;
2743:  !*         KL2 Spueleimer ;
2744:  !* (an Pneum. Schwenkeinheit KL2) ;
2745:  !*    KL2 in Ruhest. schwenken ;
2746:  !******************************** ;
2747:   ;
2748:  LBL[47] ;
2749:  R[41]=47    ;
2750:  !RSK gestartet ;
2751:  F[321]=(OFF) ;
2752:  DO[177]=(ON) ;
2753:  !Steuerluft EIN ;
2754:  DO[2121]=(ON) ;
2755:  TIMER[9]=((-2)) ;
2756:  !Warte auf Vorwahl Ventilinsel ;
2757:  WAIT ((F[523] AND !F[524]) OR (!F[523] AND F[524]) OR (TIMER[9]>=0))    ;
2758:  DO[120]=(TIMER[9]>=0) ;
2759:  DO[18181]=((TIMER[9]>=0)) ;
2760:  WAIT ((F[523] AND !F[524]) OR (!F[523] AND F[524]))    ;
2761:  DO[120]=(OFF) ;
2762:  DO[18181]=(OFF) ;
2763:  !Warte Steuerluft EIN ;
2764:  WAIT ((F[523] AND !F[524] AND DI[2121]) OR (!F[523] AND F[524] AND !DI[2122]) OR (TIMER[9]>=0))    ;
2765:  DO[120]=(TIMER[9]>=0) ;
2766:  DO[18181]=((TIMER[9]>=0)) ;
2767:  WAIT ((F[523] AND !F[524] AND DI[2121]) OR (!F[523] AND F[524] AND !DI[2122]))    ;
2768:  DO[120]=(OFF) ;
2769:  DO[18181]=(OFF) ;
2770:  !In Ruhestellung schwenken EIN ;
2771:  DO[2123]=(ON) ;
2772:  DO[2124]=(OFF) ;
2773:  !Freigabe Bewegung EIN ;
2774:  DO[2125]=(OFF) ;
2775:  DO[2126]=(ON) ;
2776:  TIMER[9]=((-10)) ;
2777:  !Warte bis Spueleimer in Position ;
2778:  WAIT ((DI[2123] AND !DI[2124]) OR (TIMER[9]>=0))    ;
2779:  DO[120]=(TIMER[9]>=0) ;
2780:  DO[18181]=((TIMER[9]>=0)) ;
2781:  WAIT (DI[2123] AND !DI[2124])    ;
2782:  DO[120]=(OFF) ;
2783:  DO[18181]=(OFF) ;
2784:  F[376]=(DI[2123] AND !DI[2124]) ;
2785:  WAIT    .30(sec) ;
2786:  !In Ruhestellung schwenken AUS ;
2787:  DO[2123]=(OFF) ;
2788:  !In Arbeitsstellung schwenken AU ;
2789:  DO[2124]=(OFF) ;
2790:  !Freigabe Bewegung AUS ;
2791:  DO[2126]=(OFF) ;
2792:  TIMER[9]=((-5)) ;
2793:  WAIT (DI[2126] OR (TIMER[9]>=0))    ;
2794:  DO[120]=(TIMER[9]>=0) ;
2795:  DO[18181]=((TIMER[9]>=0)) ;
2796:  WAIT (DI[2126])    ;
2797:  DO[120]=(OFF) ;
2798:  DO[18181]=(OFF) ;
2799:  !Freigabe  in  Endlage  halten ;
2800:  DO[2125]=(ON) ;
2801:  TIMER[9]=((-10)) ;
2802:  WAIT (DI[2125] OR (TIMER[9]>=0))    ;
2803:  DO[120]=(TIMER[9]>=0) ;
2804:  DO[18181]=((TIMER[9]>=0)) ;
2805:  WAIT (DI[2125])    ;
2806:  DO[120]=(OFF) ;
2807:  DO[18181]=(OFF) ;
2808:  DO[177]=(OFF) ;
2809:  R[42]=47    ;
2810:  JMP LBL[1] ;
2811:   ;
2812:  !******************************** ;
2813:  !*            Schritt 48 ;
2814:  !*          KL3 Spueleimer ;
2815:  !*  (an Pneum. Schwenkeinheit KL3 ;
2816:  !*     KL3 in Arbeitsst. schwenke ;
2817:  !******************************** ;
2818:   ;
2819:  LBL[48] ;
2820:  R[41]=48    ;
2821:  !RSK gestartet ;
2822:  F[321]=(OFF) ;
2823:  DO[193]=(ON) ;
2824:  !Steuerluft EIN ;
2825:  DO[2129]=(ON) ;
2826:  TIMER[9]=((-2)) ;
2827:  !Warte auf Vorwahl Ventilinsel ;
2828:  WAIT ((F[523] AND !F[524]) OR (!F[523] AND F[524]) OR (TIMER[9]>=0))    ;
2829:  DO[120]=(TIMER[9]>=0) ;
2830:  DO[18181]=((TIMER[9]>=0)) ;
2831:  WAIT ((F[523] AND !F[524]) OR (!F[523] AND F[524]))    ;
2832:  DO[120]=(OFF) ;
2833:  DO[18181]=(OFF) ;
2834:  !Warte bis Steuerluft EIN ;
2835:  WAIT ((F[523] AND !F[524] AND DI[2129]) OR (!F[523] AND F[524] AND !DI[2130]) OR (TIMER[9]>=0))    ;
2836:  DO[120]=(TIMER[9]>=0) ;
2837:  DO[18181]=((TIMER[9]>=0)) ;
2838:  WAIT ((F[523] AND !F[524] AND DI[2129]) OR (!F[523] AND F[524] AND !DI[2130]))    ;
2839:  DO[120]=(OFF) ;
2840:  DO[18181]=(OFF) ;
2841:  !In Arbeitsstellung schwenken EI ;
2842:  DO[2131]=(OFF) ;
2843:  DO[2132]=(ON) ;
2844:  !Freigabe Bewegung EIN ;
2845:  DO[2133]=(OFF) ;
2846:  DO[2134]=(ON) ;
2847:  TIMER[9]=((-10)) ;
2848:  !Warte bis Spueleimer in Position ;
2849:  WAIT ((!DI[2131] AND DI[2132]) OR (TIMER[9]>=0))    ;
2850:  DO[120]=(TIMER[9]>=0) ;
2851:  DO[18181]=((TIMER[9]>=0)) ;
2852:  WAIT (!DI[2131] AND DI[2132])    ;
2853:  DO[120]=(OFF) ;
2854:  DO[18181]=(OFF) ;
2855:  F[397]=(!DI[2131] AND DI[2132]) ;
2856:  WAIT    .30(sec) ;
2857:  !In Ruhestellung schwenken AUS ;
2858:  DO[2131]=(OFF) ;
2859:  ! In Arbeitsstellung schwenken A ;
2860:  DO[2132]=(OFF) ;
2861:  !Freigabe Bewegung AUS ;
2862:  DO[2134]=(OFF) ;
2863:  TIMER[9]=((-5)) ;
2864:  WAIT (DI[2134] OR (TIMER[9]>=0))    ;
2865:  DO[120]=(TIMER[9]>=0) ;
2866:  DO[18181]=((TIMER[9]>=0)) ;
2867:  WAIT (DI[2134])    ;
2868:  DO[120]=(OFF) ;
2869:  DO[18181]=(OFF) ;
2870:  !Freigabe  in  Endlage  halten ;
2871:  DO[2133]=(ON) ;
2872:  TIMER[9]=((-10)) ;
2873:  WAIT (DI[2133] OR (TIMER[9]>=0))    ;
2874:  DO[120]=(TIMER[9]>=0) ;
2875:  DO[18181]=((TIMER[9]>=0)) ;
2876:  WAIT (DI[2133])    ;
2877:  DO[120]=(OFF) ;
2878:  DO[18181]=(OFF) ;
2879:  DO[193]=(OFF) ;
2880:  R[42]=48    ;
2881:  JMP LBL[1] ;
2882:   ;
2883:  !******************************** ;
2884:  !*           Schritt 49 ;
2885:  !*         KL3 Spueleimer ;
2886:  !* (an Pneum. Schwenkeinheit KL3) ;
2887:  !*    KL3 in Ruhest. schwenken ;
2888:  !******************************** ;
2889:   ;
2890:  LBL[49] ;
2891:  R[41]=49    ;
2892:  !RSK gestartet ;
2893:  F[321]=(OFF) ;
2894:  DO[193]=(ON) ;
2895:  !Steuerluft EIN ;
2896:  DO[2129]=(ON) ;
2897:  TIMER[9]=((-2)) ;
2898:  !Warte auf Vorwahl Ventilinsel ;
2899:  WAIT ((F[523] AND !F[524]) OR (!F[523] AND F[524]) OR (TIMER[9]>=0))    ;
2900:  DO[120]=(TIMER[9]>=0) ;
2901:  DO[18181]=((TIMER[9]>=0)) ;
2902:  WAIT ((F[523] AND !F[524]) OR (!F[523] AND F[524]))    ;
2903:  DO[120]=(OFF) ;
2904:  DO[18181]=(OFF) ;
2905:  !Warte bis Steuerluft EIN ;
2906:  WAIT ((F[523] AND !F[524] AND DI[2129]) OR (!F[523] AND F[524] AND !DI[2130]) OR (TIMER[9]>=0))    ;
2907:  DO[120]=(TIMER[9]>=0) ;
2908:  DO[18181]=((TIMER[9]>=0)) ;
2909:  WAIT ((F[523] AND !F[524] AND DI[2129]) OR (!F[523] AND F[524] AND !DI[2130]))    ;
2910:  DO[120]=(OFF) ;
2911:  DO[18181]=(OFF) ;
2912:  !In Ruhestellung schwenken EI ;
2913:  DO[2131]=(ON) ;
2914:  DO[2132]=(OFF) ;
2915:  !Freigabe Bewegung EIN ;
2916:  DO[2133]=(OFF) ;
2917:  DO[2134]=(ON) ;
2918:  TIMER[9]=((-10)) ;
2919:  !Warte bis Spueleimer in Position ;
2920:  WAIT ((DI[2131] AND !DI[2132]) OR (TIMER[9]>=0))    ;
2921:  DO[120]=(TIMER[9]>=0) ;
2922:  DO[18181]=((TIMER[9]>=0)) ;
2923:  WAIT (DI[2131] AND DI[2132])    ;
2924:  DO[120]=(OFF) ;
2925:  DO[18181]=(OFF) ;
2926:  F[397]=(DI[2131] AND !DI[2132]) ;
2927:  WAIT    .30(sec) ;
2928:  !In Ruhestellung schwenken AUS ;
2929:  DO[2131]=(OFF) ;
2930:  !In Arbeitsstellung schwenken A ;
2931:  DO[2132]=(OFF) ;
2932:  !Freigabe Bewegung AUS ;
2933:  DO[2134]=(OFF) ;
2934:  TIMER[9]=((-5)) ;
2935:  WAIT (DI[2134] OR (TIMER[9]>=0))    ;
2936:  DO[120]=(TIMER[9]>=0) ;
2937:  DO[18181]=((TIMER[9]>=0)) ;
2938:  WAIT (DI[2134])    ;
2939:  DO[120]=(OFF) ;
2940:  DO[18181]=(OFF) ;
2941:  !Freigabe  in  Endlage  halten ;
2942:  DO[2133]=(ON) ;
2943:  TIMER[9]=((-10)) ;
2944:  WAIT (DI[2133] OR (TIMER[9]>=0))    ;
2945:  DO[120]=(TIMER[9]>=0) ;
2946:  DO[18181]=((TIMER[9]>=0)) ;
2947:  WAIT (DI[2133])    ;
2948:  DO[120]=(OFF) ;
2949:  DO[18181]=(OFF) ;
2950:  DO[193]=(OFF) ;
2951:  R[42]=49    ;
2952:  JMP LBL[1] ;
2953:   ;
2954:   ;
2955:  !********************** ;
2956:  !*    MS1 Reinigung   * ;
2957:  !*     (an Pneum. )   * ;
2958:  !* Schwenkeinheit MS1 * ;
2959:  !********************** ;
2960:   ;
2961:   ;
2962:  !******************************* ;
2963:  !*         Schritt 50          * ;
2964:  !*       MS1 Reinigung         * ;
2965:  !* MS1 in Arbeitsst. schwenken * ;
2966:  !******************************* ;
2967:   ;
2968:  LBL[50] ;
2969:  R[41]=50    ;
2970:  !RSK gestartet ;
2971:  F[321]=(OFF) ;
2972:  F[323]=(OFF) ;
2973:  F[324]=(OFF) ;
2974:  F[329]=(OFF) ;
2975:  !Reinigung MS1 gestartet ;
2976:  !MS bei Reinigung ;
2977:  DO[116]=(ON) ;
2978:  !Reinigung MS1 gestartet ;
2979:  F[604]=(ON) ;
2980:  !Steuerluft EIN ;
2981:  DO[2161]=(ON) ;
2982:  DO[2163]=(OFF) ;
2983:  DO[2164]=(OFF) ;
2984:  DO[2165]=(OFF) ;
2985:  DO[2166]=(OFF) ;
2986:  DO[2167]=(OFF) ;
2987:  DO[2168]=(OFF) ;
2988:  !Ueberwachungszeit Schwenkeinheit ;
2989:  TIMER[8]=((-5)) ;
2990:  !RSK Fehlerausgabe Schwenkeinheit ;
2991:  F[323]=(!DI[2163]) ;
2992:  !RSK Sammelstoerung ;
2993:  F[329]=(F[323]) ;
2994:  !Sprung bei Fehler MS1 schwenken ;
2995:  IF ((DI[26] OR DI[27]) AND F[323]),JMP LBL[50] ;
2996:  WAIT ((!F[323] OR (TIMER[8]>=0)) AND ((F[523] AND !F[524] AND DI[2161]) OR (!F[523] AND F[524] AND !DI[2162])))    ;
2997:  !Schwenkeinheit 1 in Arbeitsstell ;
2998:  DO[2163]=(OFF) ;
2999:  DO[2164]=(!DO[2164]) ;
3000:  !FRG Bewegung EIN ;
3001:  DO[2165]=(OFF) ;
3002:  DO[2166]=(!DI[2164]) ;
3003:  DO[18181]=(ON) ;
3004:  WAIT ((DI[2164] AND !DI[2163]) OR (TIMER[8]>=0))    ;
3005:  DO[18181]=(OFF) ;
3006:  !RSK Fehlerausgabe Schwenkeinheit ;
3007:  F[324]=((!DI[2164] AND (TIMER[8]>=0)) OR F[324]) ;
3008:  !RSK Sammelstoerung ;
3009:  F[329]=(F[324]) ;
3010:  !In Ruhestellung schwenken AUS ;
3011:  DO[2163]=(OFF) ;
3012:  !In Arbeitsstellung schwenken AUS ;
3013:  DO[2164]=(OFF) ;
3014:  !FRG Bewegung AUS ;
3015:  DO[2166]=(OFF) ;
3016:  IF ((DI[26] OR DI[27]) AND F[324]),JMP LBL[50] ;
3017:  IF (!F[324] AND DI[2166]),JMP LBL[51] ;
3018:   ;
3019:  !*************************** ;
3020:  !*      Schritt 51         * ;
3021:  !*  MS1 Versetzeinheit in  * ;
3022:  !*   Arbeitsst. schwenken  * ;
3023:  !*************************** ;
3024:   ;
3025:  LBL[51] ;
3026:  R[41]=51    ;
3027:  !FRG in Endlage halten ein ;
3028:  DO[2165]=(ON) ;
3029:  DO[2164]=(OFF) ;
3030:  DO[2168]=(OFF) ;
3031:  DO[18181]=(ON) ;
3032:  WAIT (!DI[2165])    ;
3033:  DO[18181]=(OFF) ;
3034:  !Ueberwachungszeit Versetzeinheit ;
3035:  TIMER[8]=((-5)) ;
3036:  !Ueberwachungszeit Reinigung ;
3037:  TIMER[9]=((-6)) ;
3038:  !Versetzeinheit  in  Arbeitsst. ;
3039:  DO[2168]=(!DI[2168] AND F[576]) ;
3040:  IF (DO[2168] AND (TIMER[8]>=0) AND (DI[26] OR DI[27])),JMP LBL[51] ;
3041:  IF ((DI[2168] AND F[576]) OR (!DI[2168] AND !F[576])),JMP LBL[52] ;
3042:   ;
3043:   ;
3044:  !*************************** ;
3045:  !*      Schritt 52         * ;
3046:  !* MS1 Reinigung starten   * ;
3047:  !*************************** ;
3048:   ;
3049:  LBL[52] ;
3050:  R[41]=52    ;
3051:  !MS1 Reinigung i.O. ;
3052:  DO[18181]=(ON) ;
3053:  WAIT (DI[1864])    ;
3054:  DO[18181]=(OFF) ;
3055:  !MS1 Ausblasen EIN ;
3056:  DO[1870]=(ON) ;
3057:  !MS1 Reinigung starten ;
3058:  DO[1864]=(ON) ;
3059:  !Einschaltdauer Reingung ;
3060:  TIMER[7]=((R[26])) ;
3061:  !IF (!DI[1864] AND (TIMER[9]>=0) ;
3062:  DO[18181]=(ON) ;
3063:  WAIT (!DI[1864])    ;
3064:  WAIT ((TIMER[7]>=0))    ;
3065:  DO[18181]=(OFF) ;
3066:  !MS1 Reinigung beenden ;
3067:  DO[1864]=(OFF) ;
3068:  !MS1 Ausblasen AUS ;
3069:  DO[1870]=(OFF) ;
3070:  !MS1 Reinigung i.O. ;
3071:  DO[18181]=(ON) ;
3072:   ;
3073:  WAIT (DI[1864])    ;
3074:  DO[18181]=(OFF) ;
3075:  !MS1 Einspruehen EIN ;
3076:  DO[520]=(!F[574] AND F[575]) ;
3077:  DO[1871]=(F[574] AND F[575]) ;
3078:  !Einschaltdauer Einspruehen ;
3079:  TIMER[7]=((R[23])) ;
3080:  R[42]=52    ;
3081:  JMP LBL[53] ;
3082:   ;
3083:  !**************************** ;
3084:  !*        Schritt 53        * ;
3085:  !*       MS1 Reinigung      * ;
3086:  !*                          * ;
3087:  !**************************** ;
3088:   ;
3089:  LBL[53] ;
3090:  R[41]=53    ;
3091:  !MS1 Reinigung (an Pneum. Schwenk ;
3092:  F[323]=(OFF) ;
3093:  DO[2163]=(OFF) ;
3094:  DO[2164]=(OFF) ;
3095:  DO[2165]=(OFF) ;
3096:  DO[2166]=(OFF) ;
3097:  DO[2168]=(OFF) ;
3098:   ;
3099:  !Ueberwachungszeit Schwenkeinheit ;
3100:  TIMER[8]=((-7)) ;
3101:  WAIT ((TIMER[7]>=0))    ;
3102:  !MS1 Einspruehen AUS ;
3103:  DO[520]=(OFF) ;
3104:  DO[1871]=(OFF) ;
3105:  !Versetzeinheit in Ruhest. schw. ;
3106:  DO[2167]=(ON) ;
3107:  DO[2168]=(OFF) ;
3108:  !RSK Fehlerausgabe Schwenkeinheit ;
3109:  F[324]=(!DI[2164]) ;
3110:  !RSK Sammelstoerung ;
3111:  F[329]=(F[324]) ;
